   DATA[374,25] := 2.0;
   DATA[374,26] := 7.879262;
   DATA[374,27] := 144.7578;
   DATA[374,28] := 263.9067;
   DATA[374,29] := 12.03538;
   DATA[374,30] := 1.726096;
   DATA[374,31] := 1.271551;
   DATA[374,32] := 0.7345005;
   DATA[374,33] := 0.3086186;
   DATA[374,34] := 2.0;
   DATA[374,35] := 250.8972;
   DATA[374,36] := 1.617916;
   DATA[374,37] := 189.6789;
   DATA[374,38] := 0.000128152;
   DATA[374,39] := 1.0;
   DATA[375,0] := 2.625308;
   DATA[375,1] := 529.1664;
   DATA[375,2] := 2.0;
   DATA[375,3] := 2.0;
   DATA[375,4] := 262.0802;
   DATA[375,5] := 8.393553;
   DATA[375,6] := 328.0954;
   DATA[375,7] := 2.440265;
   DATA[375,8] := 2.0;
   DATA[375,9] := 2.0;
   DATA[375,10] := 2.0;
   DATA[375,11] := 19.73558;
   DATA[375,12] := 2.206322;
   DATA[375,13] := 971.9864;
   DATA[375,14] := 1.0;
   DATA[375,15] := 2.0;
   DATA[375,16] := 1.0;
   DATA[375,17] := 1.0;
   DATA[375,18] := 1.0;
   DATA[375,19] := 2.0;
   DATA[375,20] := 148.808;
   DATA[375,21] := 156.0369;
   DATA[375,22] := 1.719412;
   DATA[375,23] := 971.674;
   DATA[375,24] := 2.0;
   DATA[375,25] := 2.0;
   DATA[375,26] := 7.879262;
   DATA[375,27] := 144.7578;
   DATA[375,28] := 263.9067;
   DATA[375,29] := 12.03538;
   DATA[375,30] := 1.727634;
   DATA[375,31] := 1.287562;
   DATA[375,32] := 0.7345005;
   DATA[375,33] := 0.3086186;
   DATA[375,34] := 2.0;
   DATA[375,35] := 250.8972;
   DATA[375,36] := 1.617916;
   DATA[375,37] := 189.6789;
   DATA[375,38] := 0.000128152;
   DATA[375,39] := 1.0;
   DATA[376,0] := 2.619223;
   DATA[376,1] := 529.559;
   DATA[376,2] := 2.0;
   DATA[376,3] := 2.0;
   DATA[376,4] := 262.0802;
   DATA[376,5] := 8.393553;
   DATA[376,6] := 328.0954;
   DATA[376,7] := 2.440265;
   DATA[376,8] := 2.0;
   DATA[376,9] := 2.0;
   DATA[376,10] := 2.0;
   DATA[376,11] := 19.65875;
   DATA[376,12] := 2.206322;
   DATA[376,13] := 972.0665;
   DATA[376,14] := 1.0;
   DATA[376,15] := 2.0;
   DATA[376,16] := 1.0;
   DATA[376,17] := 1.0;
   DATA[376,18] := 1.0;
   DATA[376,19] := 2.0;
   DATA[376,20] := 148.808;
   DATA[376,21] := 156.0882;
   DATA[376,22] := 1.718002;
   DATA[376,23] := 971.3663;
   DATA[376,24] := 2.0;
   DATA[376,25] := 2.0;
   DATA[376,26] := 7.879262;
   DATA[376,27] := 144.7578;
   DATA[376,28] := 263.9067;
   DATA[376,29] := 12.03538;
   DATA[376,30] := 1.727634;
   DATA[376,31] := 1.301396;
   DATA[376,32] := 0.7353967;
   DATA[376,33] := 0.3086186;
   DATA[376,34] := 2.0;
   DATA[376,35] := 250.8972;
   DATA[376,36] := 1.617916;
   DATA[376,37] := 189.6629;
   DATA[376,38] := 0.000128152;
   DATA[376,39] := 1.0;
   DATA[377,0] := 2.612818;
   DATA[377,1] := 529.402;
   DATA[377,2] := 2.0;
   DATA[377,3] := 2.0;
   DATA[377,4] := 262.0802;
   DATA[377,5] := 8.393553;
   DATA[377,6] := 328.0954;
   DATA[377,7] := 2.440265;
   DATA[377,8] := 2.0;
   DATA[377,9] := 2.0;
   DATA[377,10] := 2.0;
   DATA[377,11] := 19.65875;
   DATA[377,12] := 2.208628;
   DATA[377,13] := 972.1466;
   DATA[377,14] := 1.0;
   DATA[377,15] := 2.0;
   DATA[377,16] := 1.0;
   DATA[377,17] := 1.0;
   DATA[377,18] := 1.0;
   DATA[377,19] := 2.0;
   DATA[377,20] := 148.808;
   DATA[377,21] := 156.1651;
   DATA[377,22] := 1.717874;
   DATA[377,23] := 971.251;
   DATA[377,24] := 2.0;
   DATA[377,25] := 2.0;
   DATA[377,26] := 7.879262;
   DATA[377,27] := 144.7578;
   DATA[377,28] := 263.9067;
   DATA[377,29] := 12.03538;
   DATA[377,30] := 1.727634;
   DATA[377,31] := 1.312028;
   DATA[377,32] := 0.7353967;
   DATA[377,33] := 0.3075297;
   DATA[377,34] := 2.0;
   DATA[377,35] := 250.8972;
   DATA[377,36] := 1.69801;
   DATA[377,37] := 189.5988;
   DATA[377,38] := 0.000128152;
   DATA[377,39] := 1.0;
   DATA[378,0] := 2.593601;
   DATA[378,1] := 529.7552;
   DATA[378,2] := 2.0;
   DATA[378,3] := 2.0;
   DATA[378,4] := 262.0802;
   DATA[378,5] := 8.393553;
   DATA[378,6] := 328.0954;
   DATA[378,7] := 2.440265;
   DATA[378,8] := 2.0;
   DATA[378,9] := 2.0;
   DATA[378,10] := 2.0;
   DATA[378,11] := 19.65875;
   DATA[378,12] := 2.209013;
   DATA[378,13] := 972.467;
   DATA[378,14] := 1.0;
   DATA[378,15] := 2.0;
   DATA[378,16] := 1.0;
   DATA[378,17] := 1.0;
   DATA[378,18] := 1.0;
   DATA[378,19] := 2.0;
   DATA[378,20] := 148.808;
   DATA[378,21] := 156.1651;
   DATA[378,22] := 1.716592;
   DATA[378,23] := 971.1741;
   DATA[378,24] := 2.0;
   DATA[378,25] := 2.0;
   DATA[378,26] := 7.879262;
   DATA[378,27] := 144.7578;
   DATA[378,28] := 263.9067;
   DATA[378,29] := 12.03538;
   DATA[378,30] := 1.727634;
   DATA[378,31] := 1.312284;
   DATA[378,32] := 0.7353967;
   DATA[378,33] := 0.306761;
   DATA[378,34] := 2.0;
   DATA[378,35] := 250.8972;
   DATA[378,36] := 1.69801;
   DATA[378,37] := 189.4386;
   DATA[378,38] := 0.000128152;
   DATA[378,39] := 1.0;
   DATA[379,0] := 2.578868;
   DATA[379,1] := 529.9907;
   DATA[379,2] := 2.0;
   DATA[379,3] := 2.0;
   DATA[379,4] := 262.0802;
   DATA[379,5] := 8.393553;
   DATA[379,6] := 328.0954;
   DATA[379,7] := 2.440265;
   DATA[379,8] := 2.0;
   DATA[379,9] := 2.0;
   DATA[379,10] := 2.0;
   DATA[379,11] := 19.72598;
   DATA[379,12] := 2.209269;
   DATA[379,13] := 972.467;
   DATA[379,14] := 1.0;
   DATA[379,15] := 2.0;
   DATA[379,16] := 1.0;
   DATA[379,17] := 1.0;
   DATA[379,18] := 1.0;
   DATA[379,19] := 2.0;
   DATA[379,20] := 148.808;
   DATA[379,21] := 156.1651;
   DATA[379,22] := 1.715439;
   DATA[379,23] := 971.4817;
   DATA[379,24] := 2.0;
   DATA[379,25] := 2.0;
   DATA[379,26] := 7.879262;
   DATA[379,27] := 144.7578;
   DATA[379,28] := 263.7465;
   DATA[379,29] := 12.03538;
   DATA[379,30] := 1.726737;
   DATA[379,31] := 1.296016;
   DATA[379,32] := 0.7353967;
   DATA[379,33] := 0.3086186;
   DATA[379,34] := 2.0;
   DATA[379,35] := 250.8972;
   DATA[379,36] := 1.69801;
   DATA[379,37] := 189.4386;
   DATA[379,38] := 0.000128152;
   DATA[379,39] := 1.0;
   DATA[380,0] := 2.561253;
   DATA[380,1] := 530.4225;
   DATA[380,2] := 2.0;
   DATA[380,3] := 2.0;
   DATA[380,4] := 262.0802;
   DATA[380,5] := 8.393553;
   DATA[380,6] := 328.0954;
   DATA[380,7] := 2.440265;
   DATA[380,8] := 2.0;
   DATA[380,9] := 2.0;
   DATA[380,10] := 2.0;
   DATA[380,11] := 19.72598;
   DATA[380,12] := 2.211959;
   DATA[380,13] := 972.7474;
   DATA[380,14] := 1.0;
   DATA[380,15] := 2.0;
   DATA[380,16] := 1.0;
   DATA[380,17] := 1.0;
   DATA[380,18] := 1.0;
   DATA[380,19] := 2.0;
   DATA[380,20] := 148.808;
   DATA[380,21] := 156.1651;
   DATA[380,22] := 1.71467;
   DATA[380,23] := 971.674;
   DATA[380,24] := 2.0;
   DATA[380,25] := 2.0;
   DATA[380,26] := 7.879262;
   DATA[380,27] := 144.7578;
   DATA[380,28] := 263.7465;
   DATA[380,29] := 12.03538;
   DATA[380,30] := 1.726737;
   DATA[380,31] := 1.284745;
   DATA[380,32] := 0.7353967;
   DATA[380,33] := 0.3086186;
   DATA[380,34] := 2.0;
   DATA[380,35] := 250.737;
   DATA[380,36] := 1.69801;
   DATA[380,37] := 189.4386;
   DATA[380,38] := 0.000128152;
   DATA[380,39] := 1.0;
   DATA[381,0] := 2.541716;
   DATA[381,1] := 530.187;
   DATA[381,2] := 2.0;
   DATA[381,3] := 2.0;
   DATA[381,4] := 262.0802;
   DATA[381,5] := 8.393553;
   DATA[381,6] := 328.0954;
   DATA[381,7] := 2.440265;
   DATA[381,8] := 2.0;
   DATA[381,9] := 2.0;
   DATA[381,10] := 2.0;
   DATA[381,11] := 19.72598;
   DATA[381,12] := 2.211959;
   DATA[381,13] := 972.6273;
   DATA[381,14] := 1.0;
   DATA[381,15] := 2.0;
   DATA[381,16] := 1.0;
   DATA[381,17] := 1.0;
   DATA[381,18] := 1.0;
   DATA[381,19] := 2.0;
   DATA[381,20] := 148.808;
   DATA[381,21] := 156.1651;
   DATA[381,22] := 1.714286;
   DATA[381,23] := 971.674;
   DATA[381,24] := 2.0;
   DATA[381,25] := 2.0;
   DATA[381,26] := 7.879262;
   DATA[381,27] := 144.7578;
   DATA[381,28] := 263.7465;
   DATA[381,29] := 12.03538;
   DATA[381,30] := 1.726737;
   DATA[381,31] := 1.282567;
   DATA[381,32] := 0.7353967;
   DATA[381,33] := 0.3075937;
   DATA[381,34] := 2.0;
   DATA[381,35] := 250.737;
   DATA[381,36] := 1.69801;
   DATA[381,37] := 189.4386;
   DATA[381,38] := 0.000128152;
   DATA[381,39] := 1.0;
   DATA[382,0] := 2.527303;
   DATA[382,1] := 530.501;
   DATA[382,2] := 2.0;
   DATA[382,3] := 2.0;
   DATA[382,4] := 262.0802;
   DATA[382,5] := 8.393553;
   DATA[382,6] := 328.2235;
   DATA[382,7] := 2.440265;
   DATA[382,8] := 2.0;
   DATA[382,9] := 2.0;
   DATA[382,10] := 2.0;
   DATA[382,11] := 19.72598;
   DATA[382,12] := 2.211959;
   DATA[382,13] := 972.5872;
   DATA[382,14] := 1.0;
   DATA[382,15] := 2.0;
   DATA[382,16] := 1.0;
   DATA[382,17] := 1.0;
   DATA[382,18] := 1.0;
   DATA[382,19] := 2.0;
   DATA[382,20] := 148.808;
   DATA[382,21] := 155.9856;
   DATA[382,22] := 1.713517;
   DATA[382,23] := 971.674;
   DATA[382,24] := 2.0;
   DATA[382,25] := 2.0;
   DATA[382,26] := 7.879262;
   DATA[382,27] := 144.7578;
   DATA[382,28] := 263.7465;
   DATA[382,29] := 12.03538;
   DATA[382,30] := 1.726737;
   DATA[382,31] := 1.296273;
   DATA[382,32] := 0.7353967;
   DATA[382,33] := 0.3068251;
   DATA[382,34] := 2.0;
   DATA[382,35] := 250.737;
   DATA[382,36] := 1.681991;
   DATA[382,37] := 189.4386;
   DATA[382,38] := 0.000128152;
   DATA[382,39] := 1.0;
   DATA[383,0] := 2.506485;
   DATA[383,1] := 530.3832;
   DATA[383,2] := 2.0;
   DATA[383,3] := 2.0;
   DATA[383,4] := 262.0802;
   DATA[383,5] := 8.393553;
   DATA[383,6] := 328.2235;
   DATA[383,7] := 2.440265;
   DATA[383,8] := 2.0;
   DATA[383,9] := 2.0;
   DATA[383,10] := 2.0;
   DATA[383,11] := 19.69396;
   DATA[383,12] := 2.211959;
   DATA[383,13] := 972.8676;
   DATA[383,14] := 1.0;
   DATA[383,15] := 2.0;
   DATA[383,16] := 1.0;
   DATA[383,17] := 1.0;
   DATA[383,18] := 1.0;
   DATA[383,19] := 2.0;
   DATA[383,20] := 148.808;
   DATA[383,21] := 155.9856;
   DATA[383,22] := 1.715824;
   DATA[383,23] := 971.8662;
   DATA[383,24] := 2.0;
   DATA[383,25] := 2.0;
   DATA[383,26] := 7.879262;
   DATA[383,27] := 144.7578;
   DATA[383,28] := 263.7465;
   DATA[383,29] := 12.03538;
   DATA[383,30] := 1.726737;
   DATA[383,31] := 1.30114;
   DATA[383,32] := 0.7353967;
   DATA[383,33] := 0.3068251;
   DATA[383,34] := 2.0;
   DATA[383,35] := 250.737;
   DATA[383,36] := 1.681991;
   DATA[383,37] := 189.5027;
   DATA[383,38] := 0.000128152;
   DATA[383,39] := 1.0;
   DATA[384,0] := 2.493995;
   DATA[384,1] := 530.4225;
   DATA[384,2] := 2.0;
   DATA[384,3] := 2.0;
   DATA[384,4] := 262.0802;
   DATA[384,5] := 8.393553;
   DATA[384,6] := 328.2235;
   DATA[384,7] := 2.440265;
   DATA[384,8] := 2.0;
   DATA[384,9] := 2.0;
   DATA[384,10] := 2.0;
   DATA[384,11] := 19.69396;
   DATA[384,12] := 2.211959;
   DATA[384,13] := 972.8275;
   DATA[384,14] := 1.0;
   DATA[384,15] := 2.0;
   DATA[384,16] := 1.0;
   DATA[384,17] := 1.0;
   DATA[384,18] := 1.0;
   DATA[384,19] := 2.0;
   DATA[384,20] := 148.808;
   DATA[384,21] := 155.9856;
   DATA[384,22] := 1.71813;
   DATA[384,23] := 971.674;
   DATA[384,24] := 2.0;
   DATA[384,25] := 2.0;
   DATA[384,26] := 7.879262;
   DATA[384,27] := 144.7578;
   DATA[384,28] := 263.7465;
   DATA[384,29] := 12.03538;
   DATA[384,30] := 1.726737;
   DATA[384,31] := 1.292174;
   DATA[384,32] := 0.7353967;
   DATA[384,33] := 0.3063127;
   DATA[384,34] := 2.0;
   DATA[384,35] := 250.8972;
   DATA[384,36] := 1.681991;
   DATA[384,37] := 189.5668;
   DATA[384,38] := 0.000128152;
   DATA[384,39] := 1.0;
   DATA[385,0] := 2.477981;
   DATA[385,1] := 529.9122;
   DATA[385,2] := 2.0;
   DATA[385,3] := 2.0;
   DATA[385,4] := 262.0802;
   DATA[385,5] := 8.390669;
   DATA[385,6] := 328.2235;
   DATA[385,7] := 2.440265;
   DATA[385,8] := 2.0;
   DATA[385,9] := 2.0;
   DATA[385,10] := 2.0;
   DATA[385,11] := 19.65555;
   DATA[385,12] := 2.212343;
   DATA[385,13] := 973.188;
   DATA[385,14] := 1.0;
   DATA[385,15] := 2.0;
   DATA[385,16] := 1.0;
   DATA[385,17] := 1.0;
   DATA[385,18] := 1.0;
   DATA[385,19] := 2.0;
   DATA[385,20] := 148.808;
   DATA[385,21] := 155.9856;
   DATA[385,22] := 1.71813;
   DATA[385,23] := 971.7509;
   DATA[385,24] := 2.0;
   DATA[385,25] := 2.0;
   DATA[385,26] := 7.879262;
   DATA[385,27] := 144.7578;
   DATA[385,28] := 263.7465;
   DATA[385,29] := 12.30454;
   DATA[385,30] := 1.726737;
   DATA[385,31] := 1.285001;
   DATA[385,32] := 0.7353967;
   DATA[385,33] := 0.3063127;
   DATA[385,34] := 2.0;
   DATA[385,35] := 250.9453;
   DATA[385,36] := 1.681991;
   DATA[385,37] := 189.5668;
   DATA[385,38] := 0.000128152;
   DATA[385,39] := 1.0;
   DATA[386,0] := 2.46549;
   DATA[386,1] := 529.7159;
   DATA[386,2] := 2.0;
   DATA[386,3] := 2.0;
   DATA[386,4] := 262.0802;
   DATA[386,5] := 8.390669;
   DATA[386,6] := 328.2235;
   DATA[386,7] := 2.440265;
   DATA[386,8] := 2.0;
   DATA[386,9] := 2.0;
   DATA[386,10] := 2.0;
   DATA[386,11] := 19.65555;
   DATA[386,12] := 2.212343;
   DATA[386,13] := 973.2681;
   DATA[386,14] := 1.0;
   DATA[386,15] := 2.0;
   DATA[386,16] := 1.0;
   DATA[386,17] := 1.0;
   DATA[386,18] := 1.0;
   DATA[386,19] := 2.0;
   DATA[386,20] := 148.808;
   DATA[386,21] := 155.9856;
   DATA[386,22] := 1.71813;
   DATA[386,23] := 971.9431;
   DATA[386,24] := 2.0;
   DATA[386,25] := 2.0;
   DATA[386,26] := 7.879262;
   DATA[386,27] := 144.7578;
   DATA[386,28] := 263.7465;
   DATA[386,29] := 12.30454;
   DATA[386,30] := 1.726737;
   DATA[386,31] := 1.27232;
   DATA[386,32] := 0.7353967;
   DATA[386,33] := 0.3068891;
   DATA[386,34] := 2.0;
   DATA[386,35] := 250.9453;
   DATA[386,36] := 1.681991;
   DATA[386,37] := 189.6949;
   DATA[386,38] := 0.000128152;
   DATA[386,39] := 1.0;
   DATA[387,0] := 2.449156;
   DATA[387,1] := 529.3234;
   DATA[387,2] := 2.0;
   DATA[387,3] := 2.0;
   DATA[387,4] := 262.0802;
   DATA[387,5] := 8.390669;
   DATA[387,6] := 328.2235;
   DATA[387,7] := 2.440265;
   DATA[387,8] := 2.0;
   DATA[387,9] := 2.0;
   DATA[387,10] := 2.0;
   DATA[387,11] := 19.65555;
   DATA[387,12] := 2.212343;
   DATA[387,13] := 973.4283;
   DATA[387,14] := 1.0;
   DATA[387,15] := 2.0;
   DATA[387,16] := 1.0;
   DATA[387,17] := 1.0;
   DATA[387,18] := 1.0;
   DATA[387,19] := 2.0;
   DATA[387,20] := 148.808;
   DATA[387,21] := 155.9856;
   DATA[387,22] := 1.71813;
   DATA[387,23] := 971.8662;
   DATA[387,24] := 2.0;
   DATA[387,25] := 2.0;
   DATA[387,26] := 7.87766;
   DATA[387,27] := 144.7578;
   DATA[387,28] := 263.7465;
   DATA[387,29] := 12.15073;
   DATA[387,30] := 1.726737;
   DATA[387,31] := 1.271551;
   DATA[387,32] := 0.7353967;
   DATA[387,33] := 0.3068891;
   DATA[387,34] := 2.0;
   DATA[387,35] := 251.0414;
   DATA[387,36] := 1.681991;
   DATA[387,37] := 189.6949;
   DATA[387,38] := 0.000128152;
   DATA[387,39] := 1.0;
   DATA[388,0] := 2.436345;
   DATA[388,1] := 528.9309;
   DATA[388,2] := 2.0;
   DATA[388,3] := 2.0;
   DATA[388,4] := 262.0802;
   DATA[388,5] := 8.390669;
   DATA[388,6] := 328.2235;
   DATA[388,7] := 2.440265;
   DATA[388,8] := 2.0;
   DATA[388,9] := 2.0;
   DATA[388,10] := 2.0;
   DATA[388,11] := 19.58832;
   DATA[388,12] := 2.212984;
   DATA[388,13] := 973.6686;
   DATA[388,14] := 1.0;
   DATA[388,15] := 2.0;
   DATA[388,16] := 1.0;
   DATA[388,17] := 1.0;
   DATA[388,18] := 1.0;
   DATA[388,19] := 2.0;
   DATA[388,20] := 148.808;
   DATA[388,21] := 155.9856;
   DATA[388,22] := 1.71813;
   DATA[388,23] := 971.9047;
   DATA[388,24] := 2.0;
   DATA[388,25] := 2.0;
   DATA[388,26] := 7.87766;
   DATA[388,27] := 144.7578;
   DATA[388,28] := 263.7465;
   DATA[388,29] := 12.15073;
   DATA[388,30] := 1.726737;
   DATA[388,31] := 1.271551;
   DATA[388,32] := 0.7353967;
   DATA[388,33] := 0.3068891;
   DATA[388,34] := 2.0;
   DATA[388,35] := 251.1055;
   DATA[388,36] := 1.681991;
   DATA[388,37] := 189.6949;
   DATA[388,38] := 0.000128152;
   DATA[388,39] := 1.0;
   DATA[389,0] := 2.425456;
   DATA[389,1] := 528.7347;
   DATA[389,2] := 2.0;
   DATA[389,3] := 2.0;
   DATA[389,4] := 262.0802;
   DATA[389,5] := 8.390669;
   DATA[389,6] := 328.2235;
   DATA[389,7] := 2.440265;
   DATA[389,8] := 2.0;
   DATA[389,9] := 2.0;
   DATA[389,10] := 2.0;
   DATA[389,11] := 19.57872;
   DATA[389,12] := 2.212984;
   DATA[389,13] := 974.1893;
   DATA[389,14] := 1.0;
   DATA[389,15] := 2.0;
   DATA[389,16] := 1.0;
   DATA[389,17] := 1.0;
   DATA[389,18] := 1.0;
   DATA[389,19] := 2.0;
   DATA[389,20] := 148.808;
   DATA[389,21] := 155.9856;
   DATA[389,22] := 1.719924;
   DATA[389,23] := 972.2892;
   DATA[389,24] := 2.0;
   DATA[389,25] := 2.0;
   DATA[389,26] := 7.87766;
   DATA[389,27] := 144.7578;
   DATA[389,28] := 263.7465;
   DATA[389,29] := 12.07383;
   DATA[389,30] := 1.726737;
   DATA[389,31] := 1.285513;
   DATA[389,32] := 0.7353967;
   DATA[389,33] := 0.3068891;
   DATA[389,34] := 2.0;
   DATA[389,35] := 251.1055;
   DATA[389,36] := 1.681991;
   DATA[389,37] := 189.8391;
   DATA[389,38] := 0.000128152;
   DATA[389,39] := 1.0;
   DATA[390,0] := 2.420651;
   DATA[390,1] := 528.6561;
   DATA[390,2] := 2.0;
   DATA[390,3] := 2.0;
   DATA[390,4] := 262.0802;
   DATA[390,5] := 8.390669;
   DATA[390,6] := 328.0441;
   DATA[390,7] := 2.440265;
   DATA[390,8] := 2.0;
   DATA[390,9] := 2.0;
   DATA[390,10] := 2.0;
   DATA[390,11] := 19.57872;
   DATA[390,12] := 2.212984;
   DATA[390,13] := 974.2695;
   DATA[390,14] := 1.0;
   DATA[390,15] := 2.0;
   DATA[390,16] := 1.0;
   DATA[390,17] := 1.0;
   DATA[390,18] := 1.0;
   DATA[390,19] := 2.0;
   DATA[390,20] := 148.808;
   DATA[390,21] := 155.9856;
   DATA[390,22] := 1.719924;
   DATA[390,23] := 972.5967;
   DATA[390,24] := 2.0;
   DATA[390,25] := 2.0;
   DATA[390,26] := 7.87766;
   DATA[390,27] := 144.7578;
   DATA[390,28] := 263.7465;
   DATA[390,29] := 12.03538;
   DATA[390,30] := 1.726737;
   DATA[390,31] := 1.302165;
   DATA[390,32] := 0.7353967;
   DATA[390,33] := 0.3068891;
   DATA[390,34] := 2.0;
   DATA[390,35] := 251.1055;
   DATA[390,36] := 1.681991;
   DATA[390,37] := 189.8391;
   DATA[390,38] := 0.000128152;
   DATA[390,39] := 1.0;
   DATA[391,0] := 2.428338;
   DATA[391,1] := 528.3421;
   DATA[391,2] := 2.0;
   DATA[391,3] := 2.0;
   DATA[391,4] := 262.0802;
   DATA[391,5] := 8.390669;
   DATA[391,6] := 328.0441;
   DATA[391,7] := 2.440265;
   DATA[391,8] := 2.0;
   DATA[391,9] := 2.0;
   DATA[391,10] := 2.0;
   DATA[391,11] := 19.57872;
   DATA[391,12] := 2.212984;
   DATA[391,13] := 973.7487;
   DATA[391,14] := 1.0;
   DATA[391,15] := 2.0;
   DATA[391,16] := 1.0;
   DATA[391,17] := 1.0;
   DATA[391,18] := 1.0;
   DATA[391,19] := 2.0;
   DATA[391,20] := 148.808;
   DATA[391,21] := 155.9856;
   DATA[391,22] := 1.719027;
   DATA[391,23] := 972.2892;
   DATA[391,24] := 2.0;
   DATA[391,25] := 2.0;
   DATA[391,26] := 7.87766;
   DATA[391,27] := 144.7578;
   DATA[391,28] := 263.7465;
   DATA[391,29] := 12.03538;
   DATA[391,30] := 1.726737;
   DATA[391,31] := 1.32932;
   DATA[391,32] := 0.7353967;
   DATA[391,33] := 0.3061845;
   DATA[391,34] := 2.0;
   DATA[391,35] := 251.1055;
   DATA[391,36] := 1.681991;
   DATA[391,37] := 189.8391;
   DATA[391,38] := 0.000128152;
   DATA[391,39] := 1.0;
   DATA[392,0] := 2.474778;
   DATA[392,1] := 528.0674;
   DATA[392,2] := 2.0;
   DATA[392,3] := 2.0;
   DATA[392,4] := 262.0802;
   DATA[392,5] := 8.39163;
   DATA[392,6] := 328.0441;
   DATA[392,7] := 2.440265;
   DATA[392,8] := 2.0;
   DATA[392,9] := 2.0;
   DATA[392,10] := 2.0;
   DATA[392,11] := 19.57872;
   DATA[392,12] := 2.212984;
   DATA[392,13] := 973.4684;
   DATA[392,14] := 1.0;
   DATA[392,15] := 2.0;
   DATA[392,16] := 1.0;
   DATA[392,17] := 1.0;
   DATA[392,18] := 1.0;
   DATA[392,19] := 2.0;
   DATA[392,20] := 148.808;
   DATA[392,21] := 155.9856;
   DATA[392,22] := 1.71813;
   DATA[392,23] := 972.2507;
   DATA[392,24] := 2.0;
   DATA[392,25] := 2.0;
   DATA[392,26] := 7.87766;
   DATA[392,27] := 144.8347;
   DATA[392,28] := 263.7465;
   DATA[392,29] := 12.03538;
   DATA[392,30] := 1.726737;
   DATA[392,31] := 1.332266;
   DATA[392,32] := 0.7353967;
   DATA[392,33] := 0.3070813;
   DATA[392,34] := 2.0;
   DATA[392,35] := 251.1055;
   DATA[392,36] := 1.681991;
   DATA[392,37] := 189.8391;
   DATA[392,38] := 0.000128152;
   DATA[392,39] := 1.0;
   DATA[393,0] := 2.524101;
   DATA[393,1] := 528.1459;
   DATA[393,2] := 2.0;
   DATA[393,3] := 2.0;
   DATA[393,4] := 262.0802;
   DATA[393,5] := 8.39163;
   DATA[393,6] := 328.0441;
   DATA[393,7] := 2.440265;
   DATA[393,8] := 2.0;
   DATA[393,9] := 2.0;
   DATA[393,10] := 2.0;
   DATA[393,11] := 19.66195;
   DATA[393,12] := 2.212984;
   DATA[393,13] := 973.7487;
   DATA[393,14] := 1.0;
   DATA[393,15] := 2.0;
   DATA[393,16] := 1.0;
   DATA[393,17] := 1.0;
   DATA[393,18] := 1.0;
   DATA[393,19] := 2.0;
   DATA[393,20] := 148.808;
   DATA[393,21] := 155.9856;
   DATA[393,22] := 1.71813;
   DATA[393,23] := 972.3276;
   DATA[393,24] := 2.0;
   DATA[393,25] := 2.0;
   DATA[393,26] := 7.87766;
   DATA[393,27] := 144.8603;
   DATA[393,28] := 263.7465;
   DATA[393,29] := 12.03538;
   DATA[393,30] := 1.728147;
   DATA[393,31] := 1.325221;
   DATA[393,32] := 0.7353967;
   DATA[393,33] := 0.3070813;
   DATA[393,34] := 2.0;
   DATA[393,35] := 251.1055;
   DATA[393,36] := 1.681991;
   DATA[393,37] := 189.6469;
   DATA[393,38] := 0.000128152;
   DATA[393,39] := 1.0;
   DATA[394,0] := 2.552285;
   DATA[394,1] := 527.7926;
   DATA[394,2] := 2.0;
   DATA[394,3] := 2.0;
   DATA[394,4] := 262.0802;
   DATA[394,5] := 8.39163;
   DATA[394,6] := 328.0441;
   DATA[394,7] := 2.440265;
   DATA[394,8] := 2.0;
   DATA[394,9] := 2.0;
   DATA[394,10] := 2.0;
   DATA[394,11] := 19.66195;
   DATA[394,12] := 2.212343;
   DATA[394,13] := 973.3882;
   DATA[394,14] := 1.0;
   DATA[394,15] := 2.0;
   DATA[394,16] := 1.0;
   DATA[394,17] := 1.0;
   DATA[394,18] := 1.0;
   DATA[394,19] := 2.0;
   DATA[394,20] := 148.808;
   DATA[394,21] := 155.7293;
   DATA[394,22] := 1.71813;
   DATA[394,23] := 972.0585;
   DATA[394,24] := 2.0;
   DATA[394,25] := 2.0;
   DATA[394,26] := 7.87766;
   DATA[394,27] := 144.8603;
   DATA[394,28] := 263.7465;
   DATA[394,29] := 12.03538;
   DATA[394,30] := 1.728147;
   DATA[394,31] := 1.315614;
   DATA[394,32] := 0.7353967;
   DATA[394,33] := 0.3070813;
   DATA[394,34] := 2.0;
   DATA[394,35] := 251.1055;
   DATA[394,36] := 1.681991;
   DATA[394,37] := 189.6469;
   DATA[394,38] := 0.000128152;
   DATA[394,39] := 1.0;
   DATA[395,0] := 2.593921;
   DATA[395,1] := 527.9496;
   DATA[395,2] := 2.0;
   DATA[395,3] := 2.0;
   DATA[395,4] := 262.0802;
   DATA[395,5] := 8.393873;
   DATA[395,6] := 328.0441;
   DATA[395,7] := 2.436933;
   DATA[395,8] := 2.0;
   DATA[395,9] := 2.0;
   DATA[395,10] := 2.0;
   DATA[395,11] := 19.66195;
   DATA[395,12] := 2.210678;
   DATA[395,13] := 973.949;
   DATA[395,14] := 1.0;
   DATA[395,15] := 2.0;
   DATA[395,16] := 1.0;
   DATA[395,17] := 1.0;
   DATA[395,18] := 1.0;
   DATA[395,19] := 2.0;
   DATA[395,20] := 148.808;
   DATA[395,21] := 155.7293;
   DATA[395,22] := 1.71813;
   DATA[395,23] := 972.0969;
   DATA[395,24] := 2.0;
   DATA[395,25] := 2.0;
   DATA[395,26] := 7.87798;
   DATA[395,27] := 144.8603;
   DATA[395,28] := 263.7465;
   DATA[395,29] := 12.15073;
   DATA[395,30] := 1.728531;
   DATA[395,31] := 1.285769;
   DATA[395,32] := 0.7353967;
   DATA[395,33] := 0.3084905;
   DATA[395,34] := 2.0;
   DATA[395,35] := 251.1055;
   DATA[395,36] := 1.681991;
   DATA[395,37] := 189.6469;
   DATA[395,38] := 0.000128152;
   DATA[395,39] := 1.0;
   DATA[396,0] := 2.621785;
   DATA[396,1] := 527.7534;
   DATA[396,2] := 2.0;
   DATA[396,3] := 2.0;
   DATA[396,4] := 262.0802;
   DATA[396,5] := 8.393873;
   DATA[396,6] := 328.0441;
   DATA[396,7] := 2.436933;
   DATA[396,8] := 2.0;
   DATA[396,9] := 2.0;
   DATA[396,10] := 2.0;
   DATA[396,11] := 19.71637;
   DATA[396,12] := 2.210037;
   DATA[396,13] := 974.0692;
   DATA[396,14] := 1.0;
   DATA[396,15] := 2.0;
   DATA[396,16] := 1.0;
   DATA[396,17] := 1.0;
   DATA[396,18] := 1.0;
   DATA[396,19] := 2.0;
   DATA[396,20] := 148.808;
   DATA[396,21] := 155.7293;
   DATA[396,22] := 1.71813;
   DATA[396,23] := 972.4045;
   DATA[396,24] := 2.0;
   DATA[396,25] := 2.0;
   DATA[396,26] := 7.879582;
   DATA[396,27] := 144.8603;
   DATA[396,28] := 263.7465;
   DATA[396,29] := 12.15073;
   DATA[396,30] := 1.728788;
   DATA[396,31] := 1.26758;
   DATA[396,32] := 0.7353967;
   DATA[396,33] := 0.3075297;
   DATA[396,34] := 2.0;
   DATA[396,35] := 250.9933;
   DATA[396,36] := 1.681991;
   DATA[396,37] := 189.6469;
   DATA[396,38] := 0.000128152;
   DATA[396,39] := 1.0;
   DATA[397,0] := 2.654774;
   DATA[397,1] := 527.6356;
   DATA[397,2] := 2.0;
   DATA[397,3] := 2.0;
   DATA[397,4] := 262.0802;
   DATA[397,5] := 8.393873;
   DATA[397,6] := 328.0441;
   DATA[397,7] := 2.440265;
   DATA[397,8] := 2.0;
   DATA[397,9] := 2.0;
   DATA[397,10] := 2.0;
   DATA[397,11] := 19.71637;
   DATA[397,12] := 2.210037;
   DATA[397,13] := 974.2695;
   DATA[397,14] := 1.0;
   DATA[397,15] := 2.0;
   DATA[397,16] := 1.0;
   DATA[397,17] := 1.0;
   DATA[397,18] := 1.0;
   DATA[397,19] := 2.0;
   DATA[397,20] := 148.808;
   DATA[397,21] := 155.7293;
   DATA[397,22] := 1.71813;
   DATA[397,23] := 972.443;
   DATA[397,24] := 2.0;
   DATA[397,25] := 2.0;
   DATA[397,26] := 7.879582;
   DATA[397,27] := 144.8603;
   DATA[397,28] := 263.7465;
   DATA[397,29] := 12.15073;
   DATA[397,30] := 1.729172;
   DATA[397,31] := 1.265147;
   DATA[397,32] := 0.7353967;
   DATA[397,33] := 0.3081703;
   DATA[397,34] := 2.0;
   DATA[397,35] := 250.8972;
   DATA[397,36] := 1.681991;
   DATA[397,37] := 189.6469;
   DATA[397,38] := 0.000128152;
   DATA[397,39] := 1.0;
   DATA[398,0] := 2.666944;
   DATA[398,1] := 527.8711;
   DATA[398,2] := 2.0;
   DATA[398,3] := 2.0;
   DATA[398,4] := 262.0802;
   DATA[398,5] := 8.393873;
   DATA[398,6] := 328.0441;
   DATA[398,7] := 2.440265;
   DATA[398,8] := 2.0;
   DATA[398,9] := 2.0;
   DATA[398,10] := 2.0;
   DATA[398,11] := 19.71637;
   DATA[398,12] := 2.210037;
   DATA[398,13] := 974.8702;
   DATA[398,14] := 1.0;
   DATA[398,15] := 2.0;
   DATA[398,16] := 1.0;
   DATA[398,17] := 1.0;
   DATA[398,18] := 1.0;
   DATA[398,19] := 2.0;
   DATA[398,20] := 148.808;
   DATA[398,21] := 155.7293;
   DATA[398,22] := 1.71813;
   DATA[398,23] := 972.6736;
   DATA[398,24] := 2.0;
   DATA[398,25] := 2.0;
   DATA[398,26] := 7.879582;
   DATA[398,27] := 144.8603;
   DATA[398,28] := 263.7465;
   DATA[398,29] := 12.15073;
   DATA[398,30] := 1.729172;
   DATA[398,31] := 1.280902;
   DATA[398,32] := 0.7353967;
   DATA[398,33] := 0.3087468;
   DATA[398,34] := 2.0;
   DATA[398,35] := 250.8972;
   DATA[398,36] := 1.681991;
   DATA[398,37] := 189.6469;
   DATA[398,38] := 0.000128152;
   DATA[398,39] := 1.0;
   DATA[399,0] := 2.659258;
   DATA[399,1] := 528.1459;
   DATA[399,2] := 2.0;
   DATA[399,3] := 2.0;
   DATA[399,4] := 262.0802;
   DATA[399,5] := 8.393873;
   DATA[399,6] := 328.0441;
   DATA[399,7] := 2.440265;
   DATA[399,8] := 2.0;
   DATA[399,9] := 2.0;
   DATA[399,10] := 2.0;
   DATA[399,11] := 19.68756;
   DATA[399,12] := 2.210037;
   DATA[399,13] := 974.8302;
   DATA[399,14] := 1.0;
   DATA[399,15] := 2.0;
   DATA[399,16] := 1.0;
   DATA[399,17] := 1.0;
   DATA[399,18] := 1.0;
   DATA[399,19] := 2.0;
   DATA[399,20] := 148.808;
   DATA[399,21] := 155.7293;
   DATA[399,22] := 1.716849;
   DATA[399,23] := 972.9813;
   DATA[399,24] := 2.0;
   DATA[399,25] := 2.0;
   DATA[399,26] := 7.879582;
   DATA[399,27] := 144.8603;
   DATA[399,28] := 263.7465;
   DATA[399,29] := 12.15073;
   DATA[399,30] := 1.729172;
   DATA[399,31] := 1.291149;
   DATA[399,32] := 0.7353967;
   DATA[399,33] := 0.3077219;
   DATA[399,34] := 2.0;
   DATA[399,35] := 251.0254;
   DATA[399,36] := 1.681991;
   DATA[399,37] := 189.6469;
   DATA[399,38] := 0.000128152;
   DATA[399,39] := 1.0;
   DATA[400,0] := 2.637158;
   DATA[400,1] := 527.9496;
   DATA[400,2] := 2.0;
   DATA[400,3] := 2.0;
   DATA[400,4] := 262.0802;
   DATA[400,5] := 8.393873;
   DATA[400,6] := 328.0441;
   DATA[400,7] := 2.440265;
   DATA[400,8] := 2.0;
   DATA[400,9] := 2.0;
   DATA[400,10] := 2.0;
   DATA[400,11] := 19.61393;
   DATA[400,12] := 2.209269;
   DATA[400,13] := 975.1506;
   DATA[400,14] := 1.0;
   DATA[400,15] := 2.0;
   DATA[400,16] := 1.0;
   DATA[400,17] := 1.0;
   DATA[400,18] := 1.0;
   DATA[400,19] := 2.0;
   DATA[400,20] := 148.808;
   DATA[400,21] := 155.7293;
   DATA[400,22] := 1.716849;
   DATA[400,23] := 973.2889;
   DATA[400,24] := 2.0;
   DATA[400,25] := 2.0;
   DATA[400,26] := 7.879582;
   DATA[400,27] := 144.8603;
   DATA[400,28] := 263.7465;
   DATA[400,29] := 12.15073;
   DATA[400,30] := 1.729172;
   DATA[400,31] := 1.306648;
   DATA[400,32] := 0.736421;
   DATA[400,33] := 0.3068891;
   DATA[400,34] := 2.0;
   DATA[400,35] := 251.0254;
   DATA[400,36] := 1.681991;
   DATA[400,37] := 189.727;
   DATA[400,38] := 0.000128152;
   DATA[400,39] := 1.0;
   DATA[401,0] := 2.622426;
   DATA[401,1] := 527.6748;
   DATA[401,2] := 2.0;
   DATA[401,3] := 2.0;
   DATA[401,4] := 262.0802;
   DATA[401,5] := 8.393873;
   DATA[401,6] := 328.0441;
   DATA[401,7] := 2.441803;
   DATA[401,8] := 2.0;
   DATA[401,9] := 2.0;
   DATA[401,10] := 2.0;
   DATA[401,11] := 19.55311;
   DATA[401,12] := 2.209269;
   DATA[401,13] := 975.431;
   DATA[401,14] := 1.0;
   DATA[401,15] := 2.0;
   DATA[401,16] := 1.0;
   DATA[401,17] := 1.0;
   DATA[401,18] := 1.0;
   DATA[401,19] := 2.0;
   DATA[401,20] := 148.808;
   DATA[401,21] := 155.7293;
   DATA[401,22] := 1.716849;
   DATA[401,23] := 973.2889;
   DATA[401,24] := 2.0;
   DATA[401,25] := 2.0;
   DATA[401,26] := 7.879582;
   DATA[401,27] := 144.8603;
   DATA[401,28] := 263.7465;
   DATA[401,29] := 12.15073;
   DATA[401,30] := 1.729172;
   DATA[401,31] := 1.305495;
   DATA[401,32] := 0.736421;
   DATA[401,33] := 0.3066329;
   DATA[401,34] := 2.0;
   DATA[401,35] := 251.1055;
   DATA[401,36] := 1.681991;
   DATA[401,37] := 189.727;
   DATA[401,38] := 0.000128152;
   DATA[401,39] := 1.0;
   DATA[402,0] := 2.619543;
   DATA[402,1] := 527.7926;
   DATA[402,2] := 2.0;
   DATA[402,3] := 2.0;
   DATA[402,4] := 262.0802;
   DATA[402,5] := 8.393873;
   DATA[402,6] := 328.0441;
   DATA[402,7] := 2.441803;
   DATA[402,8] := 2.0;
   DATA[402,9] := 2.0;
   DATA[402,10] := 2.0;
   DATA[402,11] := 19.55311;
   DATA[402,12] := 2.209269;
   DATA[402,13] := 975.431;
   DATA[402,14] := 1.0;
   DATA[402,15] := 2.0;
   DATA[402,16] := 1.0;
   DATA[402,17] := 1.0;
   DATA[402,18] := 1.0;
   DATA[402,19] := 2.0;
   DATA[402,20] := 148.808;
   DATA[402,21] := 155.7293;
   DATA[402,22] := 1.715952;
   DATA[402,23] := 973.6734;
   DATA[402,24] := 2.0;
   DATA[402,25] := 2.0;
   DATA[402,26] := 7.879582;
   DATA[402,27] := 144.9628;
   DATA[402,28] := 263.7465;
   DATA[402,29] := 12.15073;
   DATA[402,30] := 1.729172;
   DATA[402,31] := 1.292174;
   DATA[402,32] := 0.736421;
   DATA[402,33] := 0.3066329;
   DATA[402,34] := 2.0;
   DATA[402,35] := 251.1055;
   DATA[402,36] := 1.681991;
   DATA[402,37] := 189.727;
   DATA[402,38] := 0.000128152;
   DATA[402,39] := 1.0;
   DATA[403,0] := 2.61538;
   DATA[403,1] := 527.6748;
   DATA[403,2] := 2.0;
   DATA[403,3] := 2.0;
   DATA[403,4] := 262.0802;
   DATA[403,5] := 8.393873;
   DATA[403,6] := 328.0441;
   DATA[403,7] := 2.441803;
   DATA[403,8] := 2.0;
   DATA[403,9] := 2.0;
   DATA[403,10] := 2.0;
   DATA[403,11] := 19.47948;
   DATA[403,12] := 2.209269;
   DATA[403,13] := 975.5912;
   DATA[403,14] := 1.0;
   DATA[403,15] := 2.0;
   DATA[403,16] := 1.0;
   DATA[403,17] := 1.0;
   DATA[403,18] := 1.0;
   DATA[403,19] := 2.0;
   DATA[403,20] := 148.808;
   DATA[403,21] := 155.7293;
   DATA[403,22] := 1.715567;
   DATA[403,23] := 974.0579;
   DATA[403,24] := 2.0;
   DATA[403,25] := 2.0;
   DATA[403,26] := 7.879582;
   DATA[403,27] := 144.9628;
   DATA[403,28] := 263.7465;
   DATA[403,29] := 12.15073;
   DATA[403,30] := 1.729172;
   DATA[403,31] := 1.282311;
   DATA[403,32] := 0.7357808;
   DATA[403,33] := 0.3066329;
   DATA[403,34] := 2.0;
   DATA[403,35] := 251.1055;
   DATA[403,36] := 1.681991;
   DATA[403,37] := 189.727;
   DATA[403,38] := 0.000128152;
   DATA[403,39] := 1.0;
   DATA[404,0] := 2.603209;
   DATA[404,1] := 528.3813;
   DATA[404,2] := 2.0;
   DATA[404,3] := 2.0;
   DATA[404,4] := 262.0802;
   DATA[404,5] := 8.393873;
   DATA[404,6] := 328.0441;
   DATA[404,7] := 2.441803;
   DATA[404,8] := 2.0;
   DATA[404,9] := 2.0;
   DATA[404,10] := 2.0;
   DATA[404,11] := 19.47948;
   DATA[404,12] := 2.209269;
   DATA[404,13] := 975.6713;
   DATA[404,14] := 1.0;
   DATA[404,15] := 2.0;
   DATA[404,16] := 1.0;
   DATA[404,17] := 1.0;
   DATA[404,18] := 1.0;
   DATA[404,19] := 2.0;
   DATA[404,20] := 148.808;
   DATA[404,21] := 155.7293;
   DATA[404,22] := 1.715567;
   DATA[404,23] := 974.2502;
   DATA[404,24] := 2.0;
   DATA[404,25] := 2.0;
   DATA[404,26] := 7.879582;
   DATA[404,27] := 145.0397;
   DATA[404,28] := 263.4261;
   DATA[404,29] := 12.15073;
   DATA[404,30] := 1.729172;
   DATA[404,31] := 1.265147;
   DATA[404,32] := 0.7357808;
   DATA[404,33] := 0.3066329;
   DATA[404,34] := 2.0;
   DATA[404,35] := 251.1055;
   DATA[404,36] := 1.617916;
   DATA[404,37] := 189.727;
   DATA[404,38] := 0.000128152;
   DATA[404,39] := 1.0;
   DATA[405,0] := 2.583992;
   DATA[405,1] := 528.7347;
   DATA[405,2] := 2.0;
   DATA[405,3] := 2.0;
   DATA[405,4] := 262.0802;
   DATA[405,5] := 8.393873;
   DATA[405,6] := 328.0441;
   DATA[405,7] := 2.440778;
   DATA[405,8] := 2.0;
   DATA[405,9] := 2.0;
   DATA[405,10] := 2.0;
   DATA[405,11] := 19.51149;
   DATA[405,12] := 2.209013;
   DATA[405,13] := 975.8315;
   DATA[405,14] := 1.0;
   DATA[405,15] := 2.0;
   DATA[405,16] := 1.0;
   DATA[405,17] := 1.0;
   DATA[405,18] := 1.0;
   DATA[405,19] := 2.0;
   DATA[405,20] := 148.808;
   DATA[405,21] := 155.7293;
   DATA[405,22] := 1.717489;
   DATA[405,23] := 974.4809;
   DATA[405,24] := 2.0;
   DATA[405,25] := 2.0;
   DATA[405,26] := 7.879582;
   DATA[405,27] := 145.0397;
   DATA[405,28] := 263.4261;
   DATA[405,29] := 12.15073;
   DATA[405,30] := 1.729172;
   DATA[405,31] := 1.26694;
   DATA[405,32] := 0.7357808;
   DATA[405,33] := 0.3066329;
   DATA[405,34] := 2.0;
   DATA[405,35] := 251.1055;
   DATA[405,36] := 1.617916;
   DATA[405,37] := 189.727;
   DATA[405,38] := 0.000128152;
   DATA[405,39] := 1.0;
   DATA[406,0] := 2.568299;
   DATA[406,1] := 529.0486;
   DATA[406,2] := 2.0;
   DATA[406,3] := 2.0;
   DATA[406,4] := 262.0802;
   DATA[406,5] := 8.393873;
   DATA[406,6] := 328.0441;
   DATA[406,7] := 2.440265;
   DATA[406,8] := 2.0;
   DATA[406,9] := 2.0;
   DATA[406,10] := 2.0;
   DATA[406,11] := 19.57232;
   DATA[406,12] := 2.208628;
   DATA[406,13] := 975.9517;
   DATA[406,14] := 1.0;
   DATA[406,15] := 2.0;
   DATA[406,16] := 1.0;
   DATA[406,17] := 1.0;
   DATA[406,18] := 1.0;
   DATA[406,19] := 2.0;
   DATA[406,20] := 148.808;
   DATA[406,21] := 155.7293;
   DATA[406,22] := 1.717489;
   DATA[406,23] := 975.2499;
   DATA[406,24] := 2.0;
   DATA[406,25] := 2.0;
   DATA[406,26] := 7.879582;
   DATA[406,27] := 145.0397;
   DATA[406,28] := 263.4261;
   DATA[406,29] := 11.95847;
   DATA[406,30] := 1.729172;
   DATA[406,31] := 1.272576;
   DATA[406,32] := 0.7357808;
   DATA[406,33] := 0.3066329;
   DATA[406,34] := 2.0;
   DATA[406,35] := 251.1055;
   DATA[406,36] := 1.617916;
   DATA[406,37] := 189.727;
   DATA[406,38] := 0.000128152;
   DATA[406,39] := 1.0;
   DATA[407,0] := 2.54588;
   DATA[407,1] := 529.9122;
   DATA[407,2] := 2.0;
   DATA[407,3] := 2.0;
   DATA[407,4] := 262.0802;
   DATA[407,5] := 8.393873;
   DATA[407,6] := 328.0441;
   DATA[407,7] := 2.439753;
   DATA[407,8] := 2.0;
   DATA[407,9] := 2.0;
   DATA[407,10] := 2.0;
   DATA[407,11] := 19.62354;
   DATA[407,12] := 2.208628;
   DATA[407,13] := 976.192;
   DATA[407,14] := 1.0;
   DATA[407,15] := 2.0;
   DATA[407,16] := 1.0;
   DATA[407,17] := 1.0;
   DATA[407,18] := 1.0;
   DATA[407,19] := 2.0;
   DATA[407,20] := 148.808;
   DATA[407,21] := 155.7293;
   DATA[407,22] := 1.717489;
   DATA[407,23] := 975.7498;
   DATA[407,24] := 2.0;
   DATA[407,25] := 2.0;
   DATA[407,26] := 7.879582;
   DATA[407,27] := 145.0397;
   DATA[407,28] := 263.5863;
   DATA[407,29] := 11.88157;
   DATA[407,30] := 1.726737;
   DATA[407,31] := 1.281542;
   DATA[407,32] := 0.7357808;
   DATA[407,33] := 0.3066329;
   DATA[407,34] := 2.0;
   DATA[407,35] := 250.9933;
   DATA[407,36] := 1.617916;
   DATA[407,37] := 189.727;
   DATA[407,38] := 0.000128152;
   DATA[407,39] := 1.0;
   DATA[408,0] := 2.531147;
   DATA[408,1] := 531.0113;
   DATA[408,2] := 2.0;
   DATA[408,3] := 2.0;
   DATA[408,4] := 262.0802;
   DATA[408,5] := 8.393553;
   DATA[408,6] := 328.0441;
   DATA[408,7] := 2.439496;
   DATA[408,8] := 2.0;
   DATA[408,9] := 2.0;
   DATA[408,10] := 2.0;
   DATA[408,11] := 19.62674;
   DATA[408,12] := 2.209397;
   DATA[408,13] := 976.152;
   DATA[408,14] := 1.0;
   DATA[408,15] := 2.0;
   DATA[408,16] := 1.0;
   DATA[408,17] := 1.0;
   DATA[408,18] := 1.0;
   DATA[408,19] := 2.0;
   DATA[408,20] := 148.808;
   DATA[408,21] := 155.7293;
   DATA[408,22] := 1.717489;
   DATA[408,23] := 976.2112;
   DATA[408,24] := 2.0;
   DATA[408,25] := 2.0;
   DATA[408,26] := 7.879582;
   DATA[408,27] := 145.0397;
   DATA[408,28] := 263.5863;
   DATA[408,29] := 11.88157;
   DATA[408,30] := 1.726352;
   DATA[408,31] := 1.282439;
   DATA[408,32] := 0.7357808;
   DATA[408,33] := 0.3066329;
   DATA[408,34] := 2.0;
   DATA[408,35] := 250.9132;
   DATA[408,36] := 1.730048;
   DATA[408,37] := 189.727;
   DATA[408,38] := 0.000128152;
   DATA[408,39] := 1.0;
   DATA[409,0] := 2.512891;
   DATA[409,1] := 531.6786;
   DATA[409,2] := 2.0;
   DATA[409,3] := 2.0;
   DATA[409,4] := 262.0802;
   DATA[409,5] := 8.393553;
   DATA[409,6] := 328.0441;
   DATA[409,7] := 2.439496;
   DATA[409,8] := 2.0;
   DATA[409,9] := 2.0;
   DATA[409,10] := 2.0;
   DATA[409,11] := 19.69396;
   DATA[409,12] := 2.21119;
   DATA[409,13] := 975.8716;
   DATA[409,14] := 1.0;
   DATA[409,15] := 2.0;
   DATA[409,16] := 1.0;
   DATA[409,17] := 1.0;
   DATA[409,18] := 1.0;
   DATA[409,19] := 2.0;
   DATA[409,20] := 148.808;
   DATA[409,21] := 155.7293;
   DATA[409,22] := 1.717489;
   DATA[409,23] := 976.7111;
   DATA[409,24] := 2.0;
   DATA[409,25] := 2.0;
   DATA[409,26] := 7.879582;
   DATA[409,27] := 145.0397;
   DATA[409,28] := 263.5863;
   DATA[409,29] := 12.22763;
   DATA[409,30] := 1.725327;
   DATA[409,31] := 1.282439;
   DATA[409,32] := 0.7357808;
   DATA[409,33] := 0.3066329;
   DATA[409,34] := 2.0;
   DATA[409,35] := 250.9132;
   DATA[409,36] := 1.730048;
   DATA[409,37] := 189.727;
   DATA[409,38] := 0.000128152;
   DATA[409,39] := 1.0;
   DATA[410,0] := 2.50008;
   DATA[410,1] := 532.1889;
   DATA[410,2] := 2.0;
   DATA[410,3] := 2.0;
   DATA[410,4] := 262.0802;
   DATA[410,5] := 8.39163;
   DATA[410,6] := 328.0441;
   DATA[410,7] := 2.439496;
   DATA[410,8] := 2.0;
   DATA[410,9] := 2.0;
   DATA[410,10] := 2.0;
   DATA[410,11] := 19.70677;
   DATA[410,12] := 2.21119;
   DATA[410,13] := 975.9517;
   DATA[410,14] := 1.0;
   DATA[410,15] := 2.0;
   DATA[410,16] := 1.0;
   DATA[410,17] := 1.0;
   DATA[410,18] := 1.0;
   DATA[410,19] := 2.0;
   DATA[410,20] := 148.808;
   DATA[410,21] := 155.7293;
   DATA[410,22] := 1.717489;
   DATA[410,23] := 976.6727;
   DATA[410,24] := 2.0;
   DATA[410,25] := 2.0;
   DATA[410,26] := 7.87766;
   DATA[410,27] := 145.0397;
   DATA[410,28] := 263.5863;
   DATA[410,29] := 12.22763;
   DATA[410,30] := 1.725327;
   DATA[410,31] := 1.294095;
   DATA[410,32] := 0.7357808;
   DATA[410,33] := 0.3066329;
   DATA[410,34] := 2.0;
   DATA[410,35] := 250.9132;
   DATA[410,36] := 1.730048;
   DATA[410,37] := 189.727;
   DATA[410,38] := 0.000128152;
   DATA[410,39] := 1.0;
   DATA[411,0] := 2.486308;
   DATA[411,1] := 532.5814;
   DATA[411,2] := 2.0;
   DATA[411,3] := 2.0;
   DATA[411,4] := 262.0802;
   DATA[411,5] := 8.39163;
   DATA[411,6] := 328.0441;
   DATA[411,7] := 2.441034;
   DATA[411,8] := 2.0;
   DATA[411,9] := 2.0;
   DATA[411,10] := 2.0;
   DATA[411,11] := 19.70677;
   DATA[411,12] := 2.21119;
   DATA[411,13] := 975.7915;
   DATA[411,14] := 1.0;
   DATA[411,15] := 2.0;
   DATA[411,16] := 1.0;
   DATA[411,17] := 1.0;
   DATA[411,18] := 1.0;
   DATA[411,19] := 2.0;
   DATA[411,20] := 148.808;
   DATA[411,21] := 155.7293;
   DATA[411,22] := 1.717489;
   DATA[411,23] := 976.9034;
   DATA[411,24] := 2.0;
   DATA[411,25] := 2.0;
   DATA[411,26] := 7.87766;
   DATA[411,27] := 145.0397;
   DATA[411,28] := 263.5863;
   DATA[411,29] := 12.22763;
   DATA[411,30] := 1.725327;
   DATA[411,31] := 1.297041;
   DATA[411,32] := 0.7355248;
   DATA[411,33] := 0.3066329;
   DATA[411,34] := 2.0;
   DATA[411,35] := 250.9132;
   DATA[411,36] := 1.69801;
   DATA[411,37] := 189.727;
   DATA[411,38] := 0.000128152;
   DATA[411,39] := 1.0;
   DATA[412,0] := 2.471896;
   DATA[412,1] := 532.7384;
   DATA[412,2] := 2.0;
   DATA[412,3] := 2.0;
   DATA[412,4] := 262.0802;
   DATA[412,5] := 8.39163;
   DATA[412,6] := 328.0441;
   DATA[412,7] := 2.441034;
   DATA[412,8] := 2.0;
   DATA[412,9] := 2.0;
   DATA[412,10] := 2.0;
   DATA[412,11] := 19.70677;
   DATA[412,12] := 2.210934;
   DATA[412,13] := 975.9517;
   DATA[412,14] := 1.0;
   DATA[412,15] := 2.0;
   DATA[412,16] := 1.0;
   DATA[412,17] := 1.0;
   DATA[412,18] := 1.0;
   DATA[412,19] := 2.0;
   DATA[412,20] := 148.808;
   DATA[412,21] := 155.7806;
   DATA[412,22] := 1.717489;
   DATA[412,23] := 976.5573;
   DATA[412,24] := 2.0;
   DATA[412,25] := 2.0;
   DATA[412,26] := 7.87766;
   DATA[412,27] := 145.0397;
   DATA[412,28] := 263.5863;
   DATA[412,29] := 11.92002;
   DATA[412,30] := 1.725327;
   DATA[412,31] := 1.291533;
   DATA[412,32] := 0.7351407;
   DATA[412,33] := 0.3066329;
   DATA[412,34] := 2.0;
   DATA[412,35] := 250.9132;
   DATA[412,36] := 1.617916;
   DATA[412,37] := 189.727;
   DATA[412,38] := 0.000128152;
   DATA[412,39] := 1.0;
   DATA[413,0] := 2.460045;
   DATA[413,1] := 532.3459;
   DATA[413,2] := 2.0;
   DATA[413,3] := 2.0;
   DATA[413,4] := 262.0802;
   DATA[413,5] := 8.39163;
   DATA[413,6] := 328.0441;
   DATA[413,7] := 2.441034;
   DATA[413,8] := 2.0;
   DATA[413,9] := 2.0;
   DATA[413,10] := 2.0;
   DATA[413,11] := 19.70677;
   DATA[413,12] := 2.210934;
   DATA[413,13] := 975.8315;
   DATA[413,14] := 1.0;
   DATA[413,15] := 2.0;
   DATA[413,16] := 1.0;
   DATA[413,17] := 1.0;
   DATA[413,18] := 1.0;
   DATA[413,19] := 2.0;
   DATA[413,20] := 148.808;
   DATA[413,21] := 155.7806;
   DATA[413,22] := 1.717489;
   DATA[413,23] := 977.0956;
   DATA[413,24] := 2.0;
   DATA[413,25] := 2.0;
   DATA[413,26] := 7.87766;
   DATA[413,27] := 145.0397;
   DATA[413,28] := 263.5863;
   DATA[413,29] := 11.92002;
   DATA[413,30] := 1.725327;
   DATA[413,31] := 1.281798;
   DATA[413,32] := 0.7351407;
   DATA[413,33] := 0.3081703;
   DATA[413,34] := 2.0;
   DATA[413,35] := 250.9132;
   DATA[413,36] := 1.617916;
   DATA[413,37] := 189.727;
   DATA[413,38] := 0.000128152;
   DATA[413,39] := 1.0;
   DATA[414,0] := 2.443391;
   DATA[414,1] := 532.1889;
   DATA[414,2] := 2.0;
   DATA[414,3] := 2.0;
   DATA[414,4] := 262.0802;
   DATA[414,5] := 8.39163;
   DATA[414,6] := 328.0441;
   DATA[414,7] := 2.440521;
   DATA[414,8] := 2.0;
   DATA[414,9] := 2.0;
   DATA[414,10] := 2.0;
   DATA[414,11] := 19.70677;
   DATA[414,12] := 2.210934;
   DATA[414,13] := 975.7915;
   DATA[414,14] := 1.0;
   DATA[414,15] := 2.0;
   DATA[414,16] := 1.0;
   DATA[414,17] := 1.0;
   DATA[414,18] := 1.0;
   DATA[414,19] := 2.0;
   DATA[414,20] := 148.808;
   DATA[414,21] := 155.7806;
   DATA[414,22] := 1.717489;
   DATA[414,23] := 976.9803;
   DATA[414,24] := 2.0;
   DATA[414,25] := 2.0;
   DATA[414,26] := 7.87766;
   DATA[414,27] := 145.0397;
   DATA[414,28] := 263.5863;
   DATA[414,29] := 11.92002;
   DATA[414,30] := 1.725327;
   DATA[414,31] := 1.273216;
   DATA[414,32] := 0.7351407;
   DATA[414,33] := 0.3081703;
   DATA[414,34] := 2.0;
   DATA[414,35] := 250.9132;
   DATA[414,36] := 1.617916;
   DATA[414,37] := 189.727;
   DATA[414,38] := 0.000128152;
   DATA[414,39] := 1.0;
   DATA[415,0] := 2.434423;
   DATA[415,1] := 531.8749;
   DATA[415,2] := 2.0;
   DATA[415,3] := 2.0;
   DATA[415,4] := 262.0802;
   DATA[415,5] := 8.391951;
   DATA[415,6] := 328.0441;
   DATA[415,7] := 2.440521;
   DATA[415,8] := 2.0;
   DATA[415,9] := 2.0;
   DATA[415,10] := 2.0;
   DATA[415,11] := 19.76759;
   DATA[415,12] := 2.210934;
   DATA[415,13] := 975.5912;
   DATA[415,14] := 1.0;
   DATA[415,15] := 2.0;
   DATA[415,16] := 1.0;
   DATA[415,17] := 1.0;
   DATA[415,18] := 1.0;
   DATA[415,19] := 2.0;
   DATA[415,20] := 148.808;
   DATA[415,21] := 155.7806;
   DATA[415,22] := 1.717489;
   DATA[415,23] := 977.5186;
   DATA[415,24] := 2.0;
   DATA[415,25] := 2.0;
   DATA[415,26] := 7.87766;
   DATA[415,27] := 145.0397;
   DATA[415,28] := 263.5863;
   DATA[415,29] := 11.92002;
   DATA[415,30] := 1.725327;
   DATA[415,31] := 1.271551;
   DATA[415,32] := 0.7351407;
   DATA[415,33] := 0.3081703;
   DATA[415,34] := 2.0;
   DATA[415,35] := 250.9132;
   DATA[415,36] := 1.617916;
   DATA[415,37] := 189.727;
   DATA[415,38] := 0.000128152;
   DATA[415,39] := 1.0;
   DATA[416,0] := 2.426416;
   DATA[416,1] := 531.1291;
   DATA[416,2] := 2.0;
   DATA[416,3] := 2.0;
   DATA[416,4] := 262.0802;
   DATA[416,5] := 8.393232;
   DATA[416,6] := 328.0441;
   DATA[416,7] := 2.439625;
   DATA[416,8] := 2.0;
   DATA[416,9] := 2.0;
   DATA[416,10] := 2.0;
   DATA[416,11] := 19.7804;
   DATA[416,12] := 2.21055;
   DATA[416,13] := 975.6313;
   DATA[416,14] := 1.0;
   DATA[416,15] := 2.0;
   DATA[416,16] := 1.0;
   DATA[416,17] := 1.0;
   DATA[416,18] := 1.0;
   DATA[416,19] := 2.0;
   DATA[416,20] := 148.808;
   DATA[416,21] := 155.7806;
   DATA[416,22] := 1.717489;
   DATA[416,23] := 977.557;
   DATA[416,24] := 2.0;
   DATA[416,25] := 2.0;
   DATA[416,26] := 7.87766;
   DATA[416,27] := 145.0397;
   DATA[416,28] := 263.5863;
   DATA[416,29] := 11.92002;
   DATA[416,30] := 1.725327;
   DATA[416,31] := 1.275906;
   DATA[416,32] := 0.7351407;
   DATA[416,33] := 0.3083624;
   DATA[416,34] := 2.0;
   DATA[416,35] := 250.9132;
   DATA[416,36] := 1.617916;
   DATA[416,37] := 189.5347;
   DATA[416,38] := 0.000128152;
   DATA[416,39] := 1.0;
   DATA[417,0] := 2.422253;
   DATA[417,1] := 530.4225;
   DATA[417,2] := 2.0;
   DATA[417,3] := 2.0;
   DATA[417,4] := 262.0802;
   DATA[417,5] := 8.393553;
   DATA[417,6] := 328.0441;
   DATA[417,7] := 2.43924;
   DATA[417,8] := 2.0;
   DATA[417,9] := 2.0;
   DATA[417,10] := 2.0;
   DATA[417,11] := 19.7804;
   DATA[417,12] := 2.210037;
   DATA[417,13] := 975.6713;
   DATA[417,14] := 1.0;
   DATA[417,15] := 2.0;
   DATA[417,16] := 1.0;
   DATA[417,17] := 1.0;
   DATA[417,18] := 1.0;
   DATA[417,19] := 2.0;
   DATA[417,20] := 148.808;
   DATA[417,21] := 155.7806;
   DATA[417,22] := 1.717489;
   DATA[417,23] := 977.4417;
   DATA[417,24] := 2.0;
   DATA[417,25] := 2.0;
   DATA[417,26] := 7.87766;
   DATA[417,27] := 145.0397;
   DATA[417,28] := 263.5863;
   DATA[417,29] := 12.15073;
   DATA[417,30] := 1.72789;
   DATA[417,31] := 1.290893;
   DATA[417,32] := 0.7351407;
   DATA[417,33] := 0.3083624;
   DATA[417,34] := 2.0;
   DATA[417,35] := 250.9132;
   DATA[417,36] := 1.617916;
   DATA[417,37] := 189.5347;
   DATA[417,38] := 0.000128152;
   DATA[417,39] := 1.0;
   DATA[418,0] := 2.428018;
   DATA[418,1] := 530.1085;
   DATA[418,2] := 2.0;
   DATA[418,3] := 2.0;
   DATA[418,4] := 262.0802;
   DATA[418,5] := 8.393553;
   DATA[418,6] := 328.0441;
   DATA[418,7] := 2.43924;
   DATA[418,8] := 2.0;
   DATA[418,9] := 2.0;
   DATA[418,10] := 2.0;
   DATA[418,11] := 19.72598;
   DATA[418,12] := 2.210037;
   DATA[418,13] := 975.3509;
   DATA[418,14] := 1.0;
   DATA[418,15] := 2.0;
   DATA[418,16] := 1.0;
   DATA[418,17] := 1.0;
   DATA[418,18] := 1.0;
   DATA[418,19] := 2.0;
   DATA[418,20] := 148.808;
   DATA[418,21] := 155.7806;
   DATA[418,22] := 1.717489;
   DATA[418,23] := 977.3648;
   DATA[418,24] := 2.0;
   DATA[418,25] := 2.0;
   DATA[418,26] := 7.87766;
   DATA[418,27] := 145.0397;
   DATA[418,28] := 263.5863;
   DATA[418,29] := 12.41989;
   DATA[418,30] := 1.72789;
   DATA[418,31] := 1.291918;
   DATA[418,32] := 0.7351407;
   DATA[418,33] := 0.3083624;
   DATA[418,34] := 2.0;
   DATA[418,35] := 250.9132;
   DATA[418,36] := 1.617916;
   DATA[418,37] := 189.5347;
   DATA[418,38] := 0.000128152;
   DATA[418,39] := 1.0;
   DATA[419,0] := 2.468052;
   DATA[419,1] := 529.7159;
   DATA[419,2] := 2.0;
   DATA[419,3] := 2.0;
   DATA[419,4] := 262.0802;
   DATA[419,5] := 8.393553;
   DATA[419,6] := 328.0441;
   DATA[419,7] := 2.43924;
   DATA[419,8] := 2.0;
   DATA[419,9] := 2.0;
   DATA[419,10] := 2.0;
   DATA[419,11] := 19.72598;
   DATA[419,12] := 2.209909;
   DATA[419,13] := 975.5912;
   DATA[419,14] := 1.0;
   DATA[419,15] := 2.0;
   DATA[419,16] := 1.0;
   DATA[419,17] := 1.0;
   DATA[419,18] := 1.0;
   DATA[419,19] := 2.0;
   DATA[419,20] := 148.808;
   DATA[419,21] := 155.7806;
   DATA[419,22] := 1.717489;
   DATA[419,23] := 977.3264;
   DATA[419,24] := 2.0;
   DATA[419,25] := 2.0;
   DATA[419,26] := 7.87766;
   DATA[419,27] := 145.0397;
   DATA[419,28] := 263.5863;
   DATA[419,29] := 12.41989;
   DATA[419,30] := 1.72789;
   DATA[419,31] := 1.301652;
   DATA[419,32] := 0.7351407;
   DATA[419,33] := 0.3083624;
   DATA[419,34] := 2.0;
   DATA[419,35] := 250.9132;
   DATA[419,36] := 1.617916;
   DATA[419,37] := 189.6949;
   DATA[419,38] := 0.000128152;
   DATA[419,39] := 1.0;
   DATA[420,0] := 2.520257;
   DATA[420,1] := 529.7159;
   DATA[420,2] := 2.0;
   DATA[420,3] := 2.0;
   DATA[420,4] := 262.0802;
   DATA[420,5] := 8.393553;
   DATA[420,6] := 328.0441;
   DATA[420,7] := 2.439753;
   DATA[420,8] := 2.0;
   DATA[420,9] := 2.0;
   DATA[420,10] := 2.0;
   DATA[420,11] := 19.72598;
   DATA[420,12] := 2.209013;
   DATA[420,13] := 975.7915;
   DATA[420,14] := 1.0;
   DATA[420,15] := 2.0;
   DATA[420,16] := 1.0;
   DATA[420,17] := 1.0;
   DATA[420,18] := 1.0;
   DATA[420,19] := 2.0;
   DATA[420,20] := 148.808;
   DATA[420,21] := 155.7806;
   DATA[420,22] := 1.717489;
   DATA[420,23] := 977.2879;
   DATA[420,24] := 2.0;
   DATA[420,25] := 2.0;
   DATA[420,26] := 7.87766;
   DATA[420,27] := 145.0397;
   DATA[420,28] := 263.5863;
   DATA[420,29] := 12.41989;
   DATA[420,30] := 1.72789;
   DATA[420,31] := 1.296401;
   DATA[420,32] := 0.7351407;
   DATA[420,33] := 0.3083624;
   DATA[420,34] := 2.0;
   DATA[420,35] := 250.9132;
   DATA[420,36] := 1.617916;
   DATA[420,37] := 189.727;
   DATA[420,38] := 0.000128152;
   DATA[420,39] := 1.0;
   DATA[421,0] := 2.559972;
   DATA[421,1] := 529.5982;
   DATA[421,2] := 2.0;
   DATA[421,3] := 2.0;
   DATA[421,4] := 262.2084;
   DATA[421,5] := 8.393553;
   DATA[421,6] := 328.2748;
   DATA[421,7] := 2.440393;
   DATA[421,8] := 2.0;
   DATA[421,9] := 2.0;
   DATA[421,10] := 2.0;
   DATA[421,11] := 19.65555;
   DATA[421,12] := 2.211831;
   DATA[421,13] := 975.7514;
   DATA[421,14] := 1.0;
   DATA[421,15] := 2.0;
   DATA[421,16] := 1.0;
   DATA[421,17] := 1.0;
   DATA[421,18] := 1.0;
   DATA[421,19] := 2.0;
   DATA[421,20] := 148.808;
   DATA[421,21] := 155.8062;
   DATA[421,22] := 1.717489;
   DATA[421,23] := 977.2879;
   DATA[421,24] := 2.0;
   DATA[421,25] := 2.0;
   DATA[421,26] := 7.87766;
   DATA[421,27] := 145.0397;
   DATA[421,28] := 263.5863;
   DATA[421,29] := 11.95847;
   DATA[421,30] := 1.72789;
   DATA[421,31] := 1.292046;
   DATA[421,32] := 0.7351407;
   DATA[421,33] := 0.3083624;
   DATA[421,34] := 2.0;
   DATA[421,35] := 250.9132;
   DATA[421,36] := 1.617916;
   DATA[421,37] := 189.727;
   DATA[421,38] := 0.000128152;
   DATA[421,39] := 1.0;
   DATA[422,0] := 2.603209;
   DATA[422,1] := 529.0486;
   DATA[422,2] := 2.0;
   DATA[422,3] := 2.0;
   DATA[422,4] := 262.2404;
   DATA[422,5] := 8.393553;
   DATA[422,6] := 328.2748;
   DATA[422,7] := 2.440778;
   DATA[422,8] := 2.0;
   DATA[422,9] := 2.0;
   DATA[422,10] := 2.0;
   DATA[422,11] := 19.65555;
   DATA[422,12] := 2.211831;
   DATA[422,13] := 975.5511;
   DATA[422,14] := 1.0;
   DATA[422,15] := 2.0;
   DATA[422,16] := 1.0;
   DATA[422,17] := 1.0;
   DATA[422,18] := 1.0;
   DATA[422,19] := 2.0;
   DATA[422,20] := 148.808;
   DATA[422,21] := 156.0625;
   DATA[422,22] := 1.717489;
   DATA[422,23] := 977.2879;
   DATA[422,24] := 2.0;
   DATA[422,25] := 2.0;
   DATA[422,26] := 7.87766;
   DATA[422,27] := 145.0397;
   DATA[422,28] := 263.5863;
   DATA[422,29] := 11.95847;
   DATA[422,30] := 1.7293;
   DATA[422,31] := 1.291405;
   DATA[422,32] := 0.7351407;
   DATA[422,33] := 0.3083624;
   DATA[422,34] := 2.0;
   DATA[422,35] := 250.9132;
   DATA[422,36] := 1.617916;
   DATA[422,37] := 189.727;
   DATA[422,38] := 0.000128152;
   DATA[422,39] := 1.0;
   DATA[423,0] := 2.632354;
   DATA[423,1] := 529.402;
   DATA[423,2] := 2.0;
   DATA[423,3] := 2.0;
   DATA[423,4] := 262.2404;
   DATA[423,5] := 8.393553;
   DATA[423,6] := 328.2748;
   DATA[423,7] := 2.441419;
   DATA[423,8] := 2.0;
   DATA[423,9] := 2.0;
   DATA[423,10] := 2.0;
   DATA[423,11] := 19.65555;
   DATA[423,12] := 2.211831;
   DATA[423,13] := 975.9918;
   DATA[423,14] := 1.0;
   DATA[423,15] := 2.0;
   DATA[423,16] := 1.0;
   DATA[423,17] := 1.0;
   DATA[423,18] := 1.0;
   DATA[423,19] := 2.0;
   DATA[423,20] := 148.808;
   DATA[423,21] := 156.0625;
   DATA[423,22] := 1.717489;
   DATA[423,23] := 977.3648;
   DATA[423,24] := 2.0;
   DATA[423,25] := 2.0;
   DATA[423,26] := 7.878621;
   DATA[423,27] := 145.0397;
   DATA[423,28] := 263.5863;
   DATA[423,29] := 11.95847;
   DATA[423,30] := 1.7293;
   DATA[423,31] := 1.291405;
   DATA[423,32] := 0.7351407;
   DATA[423,33] := 0.3083624;
   DATA[423,34] := 2.0;
   DATA[423,35] := 250.9132;
   DATA[423,36] := 1.617916;
   DATA[423,37] := 189.6629;
   DATA[423,38] := 0.000128152;
   DATA[423,39] := 1.0;
   DATA[424,0] := 2.649649;
   DATA[424,1] := 529.3627;
   DATA[424,2] := 2.0;
   DATA[424,3] := 2.0;
   DATA[424,4] := 262.2404;
   DATA[424,5] := 8.393553;
   DATA[424,6] := 327.9672;
   DATA[424,7] := 2.441419;
   DATA[424,8] := 2.0;
   DATA[424,9] := 2.0;
   DATA[424,10] := 2.0;
   DATA[424,11] := 19.66195;
   DATA[424,12] := 2.213624;
   DATA[424,13] := 976.4324;
   DATA[424,14] := 1.0;
   DATA[424,15] := 2.0;
   DATA[424,16] := 1.0;
   DATA[424,17] := 1.0;
   DATA[424,18] := 1.0;
   DATA[424,19] := 2.0;
   DATA[424,20] := 148.808;
   DATA[424,21] := 156.0625;
   DATA[424,22] := 1.717489;
   DATA[424,23] := 976.788;
   DATA[424,24] := 2.0;
   DATA[424,25] := 2.0;
   DATA[424,26] := 7.878621;
   DATA[424,27] := 145.0397;
   DATA[424,28] := 263.5863;
   DATA[424,29] := 11.95847;
   DATA[424,30] := 1.726737;
   DATA[424,31] := 1.291405;
   DATA[424,32] := 0.7351407;
   DATA[424,33] := 0.3083624;
   DATA[424,34] := 2.0;
   DATA[424,35] := 250.9132;
   DATA[424,36] := 1.617916;
   DATA[424,37] := 189.5347;
   DATA[424,38] := 0.000128152;
   DATA[424,39] := 1.0;
   DATA[425,0] := 2.66214;
   DATA[425,1] := 529.5982;
   DATA[425,2] := 2.0;
   DATA[425,3] := 2.0;
   DATA[425,4] := 262.2404;
   DATA[425,5] := 8.393553;
   DATA[425,6] := 327.9672;
   DATA[425,7] := 2.441419;
   DATA[425,8] := 2.0;
   DATA[425,9] := 2.0;
   DATA[425,10] := 2.0;
   DATA[425,11] := 19.66195;
   DATA[425,12] := 2.213624;
   DATA[425,13] := 976.4724;
   DATA[425,14] := 1.0;
   DATA[425,15] := 2.0;
   DATA[425,16] := 1.0;
   DATA[425,17] := 1.0;
   DATA[425,18] := 1.0;
   DATA[425,19] := 2.0;
   DATA[425,20] := 148.808;
   DATA[425,21] := 156.0625;
   DATA[425,22] := 1.717489;
   DATA[425,23] := 977.0956;
   DATA[425,24] := 2.0;
   DATA[425,25] := 2.0;
   DATA[425,26] := 7.878621;
   DATA[425,27] := 145.0397;
   DATA[425,28] := 263.5863;
   DATA[425,29] := 11.95847;
   DATA[425,30] := 1.726096;
   DATA[425,31] := 1.291405;
   DATA[425,32] := 0.7351407;
   DATA[425,33] := 0.3083624;
   DATA[425,34] := 2.0;
   DATA[425,35] := 250.9132;
   DATA[425,36] := 1.617916;
   DATA[425,37] := 189.5347;
   DATA[425,38] := 0.000128152;
   DATA[425,39] := 1.0;
   DATA[426,0] := 2.66214;
   DATA[426,1] := 529.5982;
   DATA[426,2] := 2.0;
   DATA[426,3] := 2.0;
   DATA[426,4] := 262.2404;
   DATA[426,5] := 8.393553;
   DATA[426,6] := 327.9672;
   DATA[426,7] := 2.441419;
   DATA[426,8] := 2.0;
   DATA[426,9] := 2.0;
   DATA[426,10] := 2.0;
   DATA[426,11] := 19.66195;
   DATA[426,12] := 2.213624;
   DATA[426,13] := 976.4724;
   DATA[426,14] := 1.0;
   DATA[426,15] := 2.0;
   DATA[426,16] := 1.0;
   DATA[426,17] := 1.0;
   DATA[426,18] := 1.0;
   DATA[426,19] := 2.0;
   DATA[426,20] := 148.808;
   DATA[426,21] := 156.0625;
   DATA[426,22] := 1.717489;
   DATA[426,23] := 977.0956;
   DATA[426,24] := 2.0;
   DATA[426,25] := 2.0;
   DATA[426,26] := 7.878621;
   DATA[426,27] := 145.0397;
   DATA[426,28] := 263.5863;
   DATA[426,29] := 11.95847;
   DATA[426,30] := 1.726096;
   DATA[426,31] := 1.291405;
   DATA[426,32] := 0.7351407;
   DATA[426,33] := 0.3083624;
   DATA[426,34] := 2.0;
   DATA[426,35] := 250.9132;
   DATA[426,36] := 1.617916;
   DATA[426,37] := 189.5347;
   DATA[426,38] := 0.000128152;
   DATA[426,39] := 1.0;
   DATA[427,0] := 2.66214;
   DATA[427,1] := 529.7159;
   DATA[427,2] := 2.0;
   DATA[427,3] := 2.0;
   DATA[427,4] := 262.2404;
   DATA[427,5] := 8.393553;
   DATA[427,6] := 327.9672;
   DATA[427,7] := 2.441419;
   DATA[427,8] := 2.0;
   DATA[427,9] := 2.0;
   DATA[427,10] := 2.0;
   DATA[427,11] := 19.66195;
   DATA[427,12] := 2.213624;
   DATA[427,13] := 976.3522;
   DATA[427,14] := 1.0;
   DATA[427,15] := 2.0;
   DATA[427,16] := 1.0;
   DATA[427,17] := 1.0;
   DATA[427,18] := 1.0;
   DATA[427,19] := 2.0;
   DATA[427,20] := 148.808;
   DATA[427,21] := 156.0625;
   DATA[427,22] := 1.717489;
   DATA[427,23] := 976.9803;
   DATA[427,24] := 2.0;
   DATA[427,25] := 2.0;
   DATA[427,26] := 7.878621;
   DATA[427,27] := 145.0397;
   DATA[427,28] := 263.5863;
   DATA[427,29] := 11.95847;
   DATA[427,30] := 1.726096;
   DATA[427,31] := 1.283464;
   DATA[427,32] := 0.7351407;
   DATA[427,33] := 0.3083624;
   DATA[427,34] := 2.0;
   DATA[427,35] := 250.9132;
   DATA[427,36] := 1.617916;
   DATA[427,37] := 189.5347;
   DATA[427,38] := 0.000128152;
   DATA[427,39] := 1.0;
   DATA[428,0] := 2.641002;
   DATA[428,1] := 529.5982;
   DATA[428,2] := 2.0;
   DATA[428,3] := 2.0;
   DATA[428,4] := 262.2404;
   DATA[428,5] := 8.393553;
   DATA[428,6] := 327.9672;
   DATA[428,7] := 2.441419;
   DATA[428,8] := 2.0;
   DATA[428,9] := 2.0;
   DATA[428,10] := 2.0;
   DATA[428,11] := 19.66195;
   DATA[428,12] := 2.213624;
   DATA[428,13] := 976.4724;
   DATA[428,14] := 1.0;
   DATA[428,15] := 2.0;
   DATA[428,16] := 1.0;
   DATA[428,17] := 1.0;
   DATA[428,18] := 1.0;
   DATA[428,19] := 2.0;
   DATA[428,20] := 148.808;
   DATA[428,21] := 156.0625;
   DATA[428,22] := 1.717489;
   DATA[428,23] := 976.9418;
   DATA[428,24] := 2.0;
   DATA[428,25] := 2.0;
   DATA[428,26] := 7.878621;
   DATA[428,27] := 145.1679;
   DATA[428,28] := 263.5863;
   DATA[428,29] := 11.95847;
   DATA[428,30] := 1.726096;
   DATA[428,31] := 1.281542;
   DATA[428,32] := 0.7351407;
   DATA[428,33] := 0.3083624;
   DATA[428,34] := 2.0;
   DATA[428,35] := 250.9132;
   DATA[428,36] := 1.617916;
   DATA[428,37] := 189.5347;
   DATA[428,38] := 0.000128152;
   DATA[428,39] := 1.0;
   DATA[429,0] := 2.629152;
   DATA[429,1] := 529.402;
   DATA[429,2] := 2.0;
   DATA[429,3] := 2.0;
   DATA[429,4] := 262.2404;
   DATA[429,5] := 8.393553;
   DATA[429,6] := 327.9672;
   DATA[429,7] := 2.441419;
   DATA[429,8] := 2.0;
   DATA[429,9] := 2.0;
   DATA[429,10] := 2.0;
   DATA[429,11] := 19.72277;
   DATA[429,12] := 2.213624;
   DATA[429,13] := 976.192;
   DATA[429,14] := 1.0;
   DATA[429,15] := 2.0;
   DATA[429,16] := 1.0;
   DATA[429,17] := 1.0;
   DATA[429,18] := 1.0;
   DATA[429,19] := 2.0;
   DATA[429,20] := 148.808;
   DATA[429,21] := 155.96;
   DATA[429,22] := 1.717489;
   DATA[429,23] := 977.2879;
   DATA[429,24] := 2.0;
   DATA[429,25] := 2.0;
   DATA[429,26] := 7.878621;
   DATA[429,27] := 145.1679;
   DATA[429,28] := 263.5863;
   DATA[429,29] := 11.95847;
   DATA[429,30] := 1.726096;
   DATA[429,31] := 1.288075;
   DATA[429,32] := 0.7351407;
   DATA[429,33] := 0.3083624;
   DATA[429,34] := 2.0;
   DATA[429,35] := 250.9132;
   DATA[429,36] := 1.617916;
   DATA[429,37] := 189.727;
   DATA[429,38] := 0.000128152;
   DATA[429,39] := 1.0;
   DATA[430,0] := 2.62723;
   DATA[430,1] := 529.402;
   DATA[430,2] := 2.0;
   DATA[430,3] := 2.0;
   DATA[430,4] := 262.2404;
   DATA[430,5] := 8.393553;
   DATA[430,6] := 327.9672;
   DATA[430,7] := 2.441419;
   DATA[430,8] := 2.0;
   DATA[430,9] := 2.0;
   DATA[430,10] := 2.0;
   DATA[430,11] := 19.73238;
   DATA[430,12] := 2.213624;
   DATA[430,13] := 976.0718;
   DATA[430,14] := 1.0;
   DATA[430,15] := 2.0;
   DATA[430,16] := 1.0;
   DATA[430,17] := 1.0;
   DATA[430,18] := 1.0;
   DATA[430,19] := 2.0;
   DATA[430,20] := 148.808;
   DATA[430,21] := 155.96;
   DATA[430,22] := 1.717489;
   DATA[430,23] := 977.0572;
   DATA[430,24] := 2.0;
   DATA[430,25] := 2.0;
   DATA[430,26] := 7.878621;
   DATA[430,27] := 145.1679;
   DATA[430,28] := 263.5863;
   DATA[430,29] := 11.95847;
   DATA[430,30] := 1.726096;
   DATA[430,31] := 1.285641;
   DATA[430,32] := 0.7360369;
   DATA[430,33] := 0.3083624;
   DATA[430,34] := 2.0;
   DATA[430,35] := 250.8652;
   DATA[430,36] := 1.617916;
   DATA[430,37] := 189.727;
   DATA[430,38] := 0.000128152;
   DATA[430,39] := 1.0;
   DATA[431,0] := 2.610896;
   DATA[431,1] := 529.8337;
   DATA[431,2] := 2.0;
   DATA[431,3] := 2.0;
   DATA[431,4] := 262.2404;
   DATA[431,5] := 8.393553;
   DATA[431,6] := 327.9672;
   DATA[431,7] := 2.441419;
   DATA[431,8] := 2.0;
   DATA[431,9] := 2.0;
   DATA[431,10] := 2.0;
   DATA[431,11] := 19.73238;
   DATA[431,12] := 2.213624;
   DATA[431,13] := 976.0318;
   DATA[431,14] := 1.0;
   DATA[431,15] := 2.0;
   DATA[431,16] := 1.0;
   DATA[431,17] := 1.0;
   DATA[431,18] := 1.0;
   DATA[431,19] := 2.0;
   DATA[431,20] := 148.808;
   DATA[431,21] := 155.96;
   DATA[431,22] := 1.717489;
   DATA[431,23] := 977.2879;
   DATA[431,24] := 2.0;
   DATA[431,25] := 2.0;
   DATA[431,26] := 7.878621;
   DATA[431,27] := 145.1679;
   DATA[431,28] := 263.5863;
   DATA[431,29] := 11.95847;
   DATA[431,30] := 1.728019;
   DATA[431,31] := 1.289484;
   DATA[431,32] := 0.7360369;
   DATA[431,33] := 0.3083624;
   DATA[431,34] := 2.0;
   DATA[431,35] := 250.8652;
   DATA[431,36] := 1.617916;
   DATA[431,37] := 189.727;
   DATA[431,38] := 0.000128152;
   DATA[431,39] := 1.0;
   DATA[432,0] := 2.588476;
   DATA[432,1] := 530.344;
   DATA[432,2] := 2.0;
   DATA[432,3] := 2.0;
   DATA[432,4] := 261.9841;
   DATA[432,5] := 8.393553;
   DATA[432,6] := 327.9672;
   DATA[432,7] := 2.439753;
   DATA[432,8] := 2.0;
   DATA[432,9] := 2.0;
   DATA[432,10] := 2.0;
   DATA[432,11] := 19.73238;
   DATA[432,12] := 2.213624;
   DATA[432,13] := 976.6727;
   DATA[432,14] := 1.0;
   DATA[432,15] := 2.0;
   DATA[432,16] := 1.0;
   DATA[432,17] := 1.0;
   DATA[432,18] := 1.0;
   DATA[432,19] := 2.0;
   DATA[432,20] := 148.808;
   DATA[432,21] := 155.96;
   DATA[432,22] := 1.717489;
   DATA[432,23] := 977.2879;
   DATA[432,24] := 2.0;
   DATA[432,25] := 2.0;
   DATA[432,26] := 7.878621;
   DATA[432,27] := 145.1679;
   DATA[432,28] := 263.5863;
   DATA[432,29] := 11.95847;
   DATA[432,30] := 1.728916;
   DATA[432,31] := 1.292686;
   DATA[432,32] := 0.7360369;
   DATA[432,33] := 0.3083624;
   DATA[432,34] := 2.0;
   DATA[432,35] := 250.8652;
   DATA[432,36] := 1.617916;
   DATA[432,37] := 189.727;
   DATA[432,38] := 0.000128152;
   DATA[432,39] := 1.0;
   DATA[433,0] := 2.567979;
   DATA[433,1] := 530.2263;
   DATA[433,2] := 2.0;
   DATA[433,3] := 2.0;
   DATA[433,4] := 261.9841;
   DATA[433,5] := 8.393553;
   DATA[433,6] := 327.9672;
   DATA[433,7] := 2.439753;
   DATA[433,8] := 2.0;
   DATA[433,9] := 2.0;
   DATA[433,10] := 2.0;
   DATA[433,11] := 19.70357;
   DATA[433,12] := 2.213624;
   DATA[433,13] := 976.7528;
   DATA[433,14] := 1.0;
   DATA[433,15] := 2.0;
   DATA[433,16] := 1.0;
   DATA[433,17] := 1.0;
   DATA[433,18] := 1.0;
   DATA[433,19] := 2.0;
   DATA[433,20] := 148.808;
   DATA[433,21] := 155.96;
   DATA[433,22] := 1.717489;
   DATA[433,23] := 977.557;
   DATA[433,24] := 2.0;
   DATA[433,25] := 2.0;
   DATA[433,26] := 7.878621;
   DATA[433,27] := 145.1679;
   DATA[433,28] := 263.5863;
   DATA[433,29] := 12.15073;
   DATA[433,30] := 1.728916;
   DATA[433,31] := 1.286153;
   DATA[433,32] := 0.7353967;
   DATA[433,33] := 0.3083624;
   DATA[433,34] := 2.0;
   DATA[433,35] := 250.8652;
   DATA[433,36] := 1.617916;
   DATA[433,37] := 189.727;
   DATA[433,38] := 0.000128152;
   DATA[433,39] := 1.0;
   DATA[434,0] := 2.553886;
   DATA[434,1] := 529.559;
   DATA[434,2] := 2.0;
   DATA[434,3] := 2.0;
   DATA[434,4] := 261.9841;
   DATA[434,5] := 8.393553;
   DATA[434,6] := 327.9672;
   DATA[434,7] := 2.439753;
   DATA[434,8] := 2.0;
   DATA[434,9] := 2.0;
   DATA[434,10] := 2.0;
   DATA[434,11] := 19.70357;
   DATA[434,12] := 2.213624;
   DATA[434,13] := 976.9531;
   DATA[434,14] := 1.0;
   DATA[434,15] := 2.0;
   DATA[434,16] := 1.0;
   DATA[434,17] := 1.0;
   DATA[434,18] := 1.0;
   DATA[434,19] := 2.0;
   DATA[434,20] := 148.808;
   DATA[434,21] := 155.96;
   DATA[434,22] := 1.717489;
   DATA[434,23] := 977.5186;
   DATA[434,24] := 2.0;
   DATA[434,25] := 2.0;
   DATA[434,26] := 7.878621;
   DATA[434,27] := 145.1679;
   DATA[434,28] := 263.5863;
   DATA[434,29] := 12.15073;
   DATA[434,30] := 1.728916;
   DATA[434,31] := 1.290765;
   DATA[434,32] := 0.7353967;
   DATA[434,33] := 0.3083624;
   DATA[434,34] := 2.0;
   DATA[434,35] := 250.8652;
   DATA[434,36] := 1.617916;
   DATA[434,37] := 189.727;
   DATA[434,38] := 0.000128152;
   DATA[434,39] := 1.0;
   DATA[435,0] := 2.535631;
   DATA[435,1] := 529.2057;
   DATA[435,2] := 2.0;
   DATA[435,3] := 2.0;
   DATA[435,4] := 261.9841;
   DATA[435,5] := 8.393553;
   DATA[435,6] := 327.9672;
   DATA[435,7] := 2.439753;
   DATA[435,8] := 2.0;
   DATA[435,9] := 2.0;
   DATA[435,10] := 2.0;
   DATA[435,11] := 19.70357;
   DATA[435,12] := 2.213624;
   DATA[435,13] := 976.9931;
   DATA[435,14] := 1.0;
   DATA[435,15] := 2.0;
   DATA[435,16] := 1.0;
   DATA[435,17] := 1.0;
   DATA[435,18] := 1.0;
   DATA[435,19] := 2.0;
   DATA[435,20] := 148.808;
   DATA[435,21] := 155.96;
   DATA[435,22] := 1.717489;
   DATA[435,23] := 977.4802;
   DATA[435,24] := 2.0;
   DATA[435,25] := 2.0;
   DATA[435,26] := 7.878621;
   DATA[435,27] := 145.1679;
   DATA[435,28] := 263.5863;
   DATA[435,29] := 12.15073;
   DATA[435,30] := 1.728916;
   DATA[435,31] := 1.292558;
   DATA[435,32] := 0.7353967;
   DATA[435,33] := 0.3083624;
   DATA[435,34] := 2.0;
   DATA[435,35] := 251.0254;
   DATA[435,36] := 1.617916;
   DATA[435,37] := 189.727;
   DATA[435,38] := 0.000128152;
   DATA[435,39] := 1.0;
   DATA[436,0] := 2.521538;
   DATA[436,1] := 528.3813;
   DATA[436,2] := 2.0;
   DATA[436,3] := 2.0;
   DATA[436,4] := 261.9841;
   DATA[436,5] := 8.393553;
   DATA[436,6] := 328.0954;
   DATA[436,7] := 2.439753;
   DATA[436,8] := 2.0;
   DATA[436,9] := 2.0;
   DATA[436,10] := 2.0;
   DATA[436,11] := 19.70357;
   DATA[436,12] := 2.212087;
   DATA[436,13] := 977.1934;
   DATA[436,14] := 1.0;
   DATA[436,15] := 2.0;
   DATA[436,16] := 1.0;
   DATA[436,17] := 1.0;
   DATA[436,18] := 1.0;
   DATA[436,19] := 2.0;
   DATA[436,20] := 148.808;
   DATA[436,21] := 155.96;
   DATA[436,22] := 1.719284;
   DATA[436,23] := 977.6339;
   DATA[436,24] := 2.0;
   DATA[436,25] := 2.0;
   DATA[436,26] := 7.878621;
   DATA[436,27] := 145.1679;
   DATA[436,28] := 263.5863;
   DATA[436,29] := 12.15073;
   DATA[436,30] := 1.728916;
   DATA[436,31] := 1.302165;
   DATA[436,32] := 0.7353967;
   DATA[436,33] := 0.3083624;
   DATA[436,34] := 2.0;
   DATA[436,35] := 251.0414;
   DATA[436,36] := 1.649953;
   DATA[436,37] := 189.727;
   DATA[436,38] := 0.000128152;
   DATA[436,39] := 1.0;
   DATA[437,0] := 2.503923;
   DATA[437,1] := 528.0281;
   DATA[437,2] := 2.0;
   DATA[437,3] := 2.0;
   DATA[437,4] := 261.9841;
   DATA[437,5] := 8.393553;
   DATA[437,6] := 328.121;
   DATA[437,7] := 2.439753;
   DATA[437,8] := 2.0;
   DATA[437,9] := 2.0;
   DATA[437,10] := 2.0;
   DATA[437,11] := 19.70357;
   DATA[437,12] := 2.212087;
   DATA[437,13] := 977.4738;
   DATA[437,14] := 1.0;
   DATA[437,15] := 2.0;
   DATA[437,16] := 1.0;
   DATA[437,17] := 1.0;
   DATA[437,18] := 1.0;
   DATA[437,19] := 2.0;
   DATA[437,20] := 148.808;
   DATA[437,21] := 155.96;
   DATA[437,22] := 1.719284;
   DATA[437,23] := 977.6339;
   DATA[437,24] := 2.0;
   DATA[437,25] := 2.0;
   DATA[437,26] := 7.878621;
   DATA[437,27] := 145.1166;
   DATA[437,28] := 263.5863;
   DATA[437,29] := 12.15073;
   DATA[437,30] := 1.728916;
   DATA[437,31] := 1.302165;
   DATA[437,32] := 0.7353967;
   DATA[437,33] := 0.3083624;
   DATA[437,34] := 2.0;
   DATA[437,35] := 251.1535;
   DATA[437,36] := 1.69801;
   DATA[437,37] := 189.8071;
   DATA[437,38] := 0.000128152;
   DATA[437,39] := 1.0;
   DATA[438,0] := 2.490472;
   DATA[438,1] := 527.6356;
   DATA[438,2] := 2.0;
   DATA[438,3] := 2.0;
   DATA[438,4] := 262.1764;
   DATA[438,5] := 8.393553;
   DATA[438,6] := 328.121;
   DATA[438,7] := 2.439753;
   DATA[438,8] := 2.0;
   DATA[438,9] := 2.0;
   DATA[438,10] := 2.0;
   DATA[438,11] := 19.61393;
   DATA[438,12] := 2.21119;
   DATA[438,13] := 977.1533;
   DATA[438,14] := 1.0;
   DATA[438,15] := 2.0;
   DATA[438,16] := 1.0;
   DATA[438,17] := 1.0;
   DATA[438,18] := 1.0;
   DATA[438,19] := 2.0;
   DATA[438,20] := 148.808;
   DATA[438,21] := 155.96;
   DATA[438,22] := 1.719284;
   DATA[438,23] := 977.4802;
   DATA[438,24] := 2.0;
   DATA[438,25] := 2.0;
   DATA[438,26] := 7.878621;
   DATA[438,27] := 145.1166;
   DATA[438,28] := 263.362;
   DATA[438,29] := 12.15073;
   DATA[438,30] := 1.731351;
   DATA[438,31] := 1.302165;
   DATA[438,32] := 0.7353967;
   DATA[438,33] := 0.3083624;
   DATA[438,34] := 2.0;
   DATA[438,35] := 251.2817;
   DATA[438,36] := 1.69801;
   DATA[438,37] := 189.9673;
   DATA[438,38] := 0.000128152;
   DATA[438,39] := 1.0;
   DATA[439,0] := 2.473817;
   DATA[439,1] := 527.0861;
   DATA[439,2] := 2.0;
   DATA[439,3] := 2.0;
   DATA[439,4] := 262.1764;
   DATA[439,5] := 8.393553;
   DATA[439,6] := 328.121;
   DATA[439,7] := 2.439753;
   DATA[439,8] := 2.0;
   DATA[439,9] := 2.0;
   DATA[439,10] := 2.0;
   DATA[439,11] := 19.61393;
   DATA[439,12] := 2.210934;
   DATA[439,13] := 976.8729;
   DATA[439,14] := 1.0;
   DATA[439,15] := 2.0;
   DATA[439,16] := 1.0;
   DATA[439,17] := 1.0;
   DATA[439,18] := 1.0;
   DATA[439,19] := 2.0;
   DATA[439,20] := 148.808;
   DATA[439,21] := 155.96;
   DATA[439,22] := 1.719284;
   DATA[439,23] := 977.4802;
   DATA[439,24] := 2.0;
   DATA[439,25] := 2.0;
   DATA[439,26] := 7.878621;
   DATA[439,27] := 145.1166;
   DATA[439,28] := 263.362;
   DATA[439,29] := 12.15073;
   DATA[439,30] := 1.731351;
   DATA[439,31] := 1.302165;
   DATA[439,32] := 0.7353967;
   DATA[439,33] := 0.3083624;
   DATA[439,34] := 2.0;
   DATA[439,35] := 251.2817;
   DATA[439,36] := 1.69801;
   DATA[439,37] := 189.9673;
   DATA[439,38] := 0.000128152;
   DATA[439,39] := 1.0;
   DATA[440,0] := 2.461967;
   DATA[440,1] := 526.4188;
   DATA[440,2] := 2.0;
   DATA[440,3] := 2.0;
   DATA[440,4] := 262.1764;
   DATA[440,5] := 8.393553;
   DATA[440,6] := 328.121;
   DATA[440,7] := 2.439753;
   DATA[440,8] := 2.0;
   DATA[440,9] := 2.0;
   DATA[440,10] := 2.0;
   DATA[440,11] := 19.5435;
   DATA[440,12] := 2.210934;
   DATA[440,13] := 976.8329;
   DATA[440,14] := 1.0;
   DATA[440,15] := 2.0;
   DATA[440,16] := 1.0;
   DATA[440,17] := 1.0;
   DATA[440,18] := 1.0;
   DATA[440,19] := 2.0;
   DATA[440,20] := 148.808;
   DATA[440,21] := 155.96;
   DATA[440,22] := 1.720053;
   DATA[440,23] := 977.4417;
   DATA[440,24] := 2.0;
   DATA[440,25] := 2.0;
   DATA[440,26] := 7.878621;
   DATA[440,27] := 145.1166;
   DATA[440,28] := 263.362;
   DATA[440,29] := 12.15073;
   DATA[440,30] := 1.731351;
   DATA[440,31] := 1.293326;
   DATA[440,32] := 0.7353967;
   DATA[440,33] := 0.3070813;
   DATA[440,34] := 2.0;
   DATA[440,35] := 251.2817;
   DATA[440,36] := 1.69801;
   DATA[440,37] := 189.9673;
   DATA[440,38] := 0.000128152;
   DATA[440,39] := 1.0;
   DATA[441,0] := 2.446594;
   DATA[441,1] := 526.1047;
   DATA[441,2] := 2.0;
   DATA[441,3] := 2.0;
   DATA[441,4] := 262.1764;
   DATA[441,5] := 8.393553;
   DATA[441,6] := 328.121;
   DATA[441,7] := 2.439753;
   DATA[441,8] := 2.0;
   DATA[441,9] := 2.0;
   DATA[441,10] := 2.0;
   DATA[441,11] := 19.5435;
   DATA[441,12] := 2.210934;
   DATA[441,13] := 976.6727;
   DATA[441,14] := 1.0;
   DATA[441,15] := 2.0;
   DATA[441,16] := 1.0;
   DATA[441,17] := 1.0;
   DATA[441,18] := 1.0;
   DATA[441,19] := 2.0;
   DATA[441,20] := 148.808;
   DATA[441,21] := 155.96;
   DATA[441,22] := 1.720565;
   DATA[441,23] := 977.6724;
   DATA[441,24] := 2.0;
   DATA[441,25] := 2.0;
   DATA[441,26] := 7.878621;
   DATA[441,27] := 145.1166;
   DATA[441,28] := 263.362;
   DATA[441,29] := 11.95847;
   DATA[441,30] := 1.731351;
   DATA[441,31] := 1.308185;
   DATA[441,32] := 0.7353967;
   DATA[441,33] := 0.3068251;
   DATA[441,34] := 2.0;
   DATA[441,35] := 251.2817;
   DATA[441,36] := 1.69801;
   DATA[441,37] := 189.9673;
   DATA[441,38] := 0.000128152;
   DATA[441,39] := 1.0;
   DATA[442,0] := 2.425776;
   DATA[442,1] := 526.458;
   DATA[442,2] := 2.0;
   DATA[442,3] := 2.0;
   DATA[442,4] := 262.1764;
   DATA[442,5] := 8.393553;
   DATA[442,6] := 328.121;
   DATA[442,7] := 2.439753;
   DATA[442,8] := 2.0;
   DATA[442,9] := 2.0;
   DATA[442,10] := 2.0;
   DATA[442,11] := 19.5435;
   DATA[442,12] := 2.210934;
   DATA[442,13] := 977.2334;
   DATA[442,14] := 1.0;
   DATA[442,15] := 2.0;
   DATA[442,16] := 1.0;
   DATA[442,17] := 1.0;
   DATA[442,18] := 1.0;
   DATA[442,19] := 2.0;
   DATA[442,20] := 148.808;
   DATA[442,21] := 155.96;
   DATA[442,22] := 1.720565;
   DATA[442,23] := 977.4802;
   DATA[442,24] := 2.0;
   DATA[442,25] := 2.0;
   DATA[442,26] := 7.878621;
   DATA[442,27] := 145.1166;
   DATA[442,28] := 263.362;
   DATA[442,29] := 11.95847;
   DATA[442,30] := 1.731351;
   DATA[442,31] := 1.310747;
   DATA[442,32] := 0.7353967;
   DATA[442,33] := 0.3068251;
   DATA[442,34] := 2.0;
   DATA[442,35] := 251.2817;
   DATA[442,36] := 1.69801;
   DATA[442,37] := 189.9673;
   DATA[442,38] := 0.000128152;
   DATA[442,39] := 1.0;
   DATA[443,0] := 2.420011;
   DATA[443,1] := 527.2038;
   DATA[443,2] := 2.0;
   DATA[443,3] := 2.0;
   DATA[443,4] := 262.1764;
   DATA[443,5] := 8.393553;
   DATA[443,6] := 327.9928;
   DATA[443,7] := 2.439753;
   DATA[443,8] := 2.0;
   DATA[443,9] := 2.0;
   DATA[443,10] := 2.0;
   DATA[443,11] := 19.57232;
   DATA[443,12] := 2.208244;
   DATA[443,13] := 977.0732;
   DATA[443,14] := 1.0;
   DATA[443,15] := 2.0;
   DATA[443,16] := 1.0;
   DATA[443,17] := 1.0;
   DATA[443,18] := 1.0;
   DATA[443,19] := 2.0;
   DATA[443,20] := 148.808;
   DATA[443,21] := 155.96;
   DATA[443,22] := 1.720565;
   DATA[443,23] := 977.7493;
   DATA[443,24] := 2.0;
   DATA[443,25] := 2.0;
   DATA[443,26] := 7.878621;
   DATA[443,27] := 145.1166;
   DATA[443,28] := 263.362;
   DATA[443,29] := 11.95847;
   DATA[443,30] := 1.731351;
   DATA[443,31] := 1.302165;
   DATA[443,32] := 0.7353967;
   DATA[443,33] := 0.3068251;
   DATA[443,34] := 2.0;
   DATA[443,35] := 251.2817;
   DATA[443,36] := 1.69801;
   DATA[443,37] := 189.9673;
   DATA[443,38] := 0.000128152;
   DATA[443,39] := 1.0;
   DATA[444,0] := 2.417769;
   DATA[444,1] := 527.7926;
   DATA[444,2] := 2.0;
   DATA[444,3] := 2.0;
   DATA[444,4] := 262.1764;
   DATA[444,5] := 8.393553;
   DATA[444,6] := 327.9928;
   DATA[444,7] := 2.439753;
   DATA[444,8] := 2.0;
   DATA[444,9] := 2.0;
   DATA[444,10] := 2.0;
   DATA[444,11] := 19.59472;
   DATA[444,12] := 2.207603;
   DATA[444,13] := 976.9931;
   DATA[444,14] := 1.0;
   DATA[444,15] := 2.0;
   DATA[444,16] := 1.0;
   DATA[444,17] := 1.0;
   DATA[444,18] := 1.0;
   DATA[444,19] := 2.0;
   DATA[444,20] := 148.808;
   DATA[444,21] := 155.8575;
   DATA[444,22] := 1.720565;
   DATA[444,23] := 977.7108;
   DATA[444,24] := 2.0;
   DATA[444,25] := 2.0;
   DATA[444,26] := 7.878621;
   DATA[444,27] := 145.1166;
   DATA[444,28] := 263.362;
   DATA[444,29] := 11.95847;
   DATA[444,30] := 1.731351;
   DATA[444,31] := 1.29512;
   DATA[444,32] := 0.7353967;
   DATA[444,33] := 0.3068251;
   DATA[444,34] := 2.0;
   DATA[444,35] := 251.2817;
   DATA[444,36] := 1.69801;
   DATA[444,37] := 189.9673;
   DATA[444,38] := 0.000128152;
   DATA[444,39] := 1.0;
   DATA[445,0] := 2.417769;
   DATA[445,1] := 527.7926;
   DATA[445,2] := 2.0;
   DATA[445,3] := 2.0;
   DATA[445,4] := 262.1764;
   DATA[445,5] := 8.393553;
   DATA[445,6] := 327.9928;
   DATA[445,7] := 2.439753;
   DATA[445,8] := 2.0;
   DATA[445,9] := 2.0;
   DATA[445,10] := 2.0;
   DATA[445,11] := 19.59472;
   DATA[445,12] := 2.206835;
   DATA[445,13] := 977.4337;
   DATA[445,14] := 1.0;
   DATA[445,15] := 2.0;
   DATA[445,16] := 1.0;
   DATA[445,17] := 1.0;
   DATA[445,18] := 1.0;
   DATA[445,19] := 2.0;
   DATA[445,20] := 148.808;
   DATA[445,21] := 155.8318;
   DATA[445,22] := 1.720565;
   DATA[445,23] := 977.557;
   DATA[445,24] := 2.0;
   DATA[445,25] := 2.0;
   DATA[445,26] := 7.878621;
   DATA[445,27] := 145.1166;
   DATA[445,28] := 263.362;
   DATA[445,29] := 11.95847;
   DATA[445,30] := 1.731351;
   DATA[445,31] := 1.291277;
   DATA[445,32] := 0.7353967;
   DATA[445,33] := 0.3068251;
   DATA[445,34] := 2.0;
   DATA[445,35] := 251.2817;
   DATA[445,36] := 1.69801;
   DATA[445,37] := 189.9673;
   DATA[445,38] := 0.000128152;
   DATA[445,39] := 1.0;
   DATA[446,0] := 2.471575;
   DATA[446,1] := 528.2244;
   DATA[446,2] := 2.0;
   DATA[446,3] := 2.0;
   DATA[446,4] := 262.1764;
   DATA[446,5] := 8.393553;
   DATA[446,6] := 327.9928;
   DATA[446,7] := 2.439753;
   DATA[446,8] := 2.0;
   DATA[446,9] := 2.0;
   DATA[446,10] := 2.0;
   DATA[446,11] := 19.59472;
   DATA[446,12] := 2.206835;
   DATA[446,13] := 977.0732;
   DATA[446,14] := 1.0;
   DATA[446,15] := 2.0;
   DATA[446,16] := 1.0;
   DATA[446,17] := 1.0;
   DATA[446,18] := 1.0;
   DATA[446,19] := 2.0;
   DATA[446,20] := 148.808;
   DATA[446,21] := 155.8318;
   DATA[446,22] := 1.719284;
   DATA[446,23] := 977.2879;
   DATA[446,24] := 2.0;
   DATA[446,25] := 2.0;
   DATA[446,26] := 7.878621;
   DATA[446,27] := 145.1166;
   DATA[446,28] := 263.362;
   DATA[446,29] := 11.95847;
   DATA[446,30] := 1.731351;
   DATA[446,31] := 1.291277;
   DATA[446,32] := 0.7353967;
   DATA[446,33] := 0.3068251;
   DATA[446,34] := 2.0;
   DATA[446,35] := 251.2817;
   DATA[446,36] := 1.69801;
   DATA[446,37] := 189.9673;
   DATA[446,38] := 0.000128152;
   DATA[446,39] := 1.0;
   DATA[447,0] := 2.518336;
   DATA[447,1] := 528.5776;
   DATA[447,2] := 2.0;
   DATA[447,3] := 2.0;
   DATA[447,4] := 262.1764;
   DATA[447,5] := 8.393553;
   DATA[447,6] := 327.9928;
   DATA[447,7] := 2.439753;
   DATA[447,8] := 2.0;
   DATA[447,9] := 2.0;
   DATA[447,10] := 2.0;
   DATA[447,11] := 19.66835;
   DATA[447,12] := 2.206835;
   DATA[447,13] := 977.634;
   DATA[447,14] := 1.0;
   DATA[447,15] := 2.0;
   DATA[447,16] := 1.0;
   DATA[447,17] := 1.0;
   DATA[447,18] := 1.0;
   DATA[447,19] := 2.0;
   DATA[447,20] := 148.808;
   DATA[447,21] := 155.8575;
   DATA[447,22] := 1.718771;
   DATA[447,23] := 977.2879;
   DATA[447,24] := 2.0;
   DATA[447,25] := 2.0;
   DATA[447,26] := 7.878621;
   DATA[447,27] := 145.1166;
   DATA[447,28] := 263.362;
   DATA[447,29] := 11.95847;
   DATA[447,30] := 1.731351;
   DATA[447,31] := 1.302037;
   DATA[447,32] := 0.7353967;
   DATA[447,33] := 0.3068251;
   DATA[447,34] := 2.0;
   DATA[447,35] := 251.2817;
   DATA[447,36] := 1.69801;
   DATA[447,37] := 189.9673;
   DATA[447,38] := 0.000128152;
   DATA[447,39] := 1.0;
   DATA[448,0] := 2.558691;
   DATA[448,1] := 529.2057;
   DATA[448,2] := 2.0;
   DATA[448,3] := 2.0;
   DATA[448,4] := 262.1764;
   DATA[448,5] := 8.394835;
   DATA[448,6] := 327.9928;
   DATA[448,7] := 2.439753;
   DATA[448,8] := 2.0;
   DATA[448,9] := 2.0;
   DATA[448,10] := 2.0;
   DATA[448,11] := 19.66835;
   DATA[448,12] := 2.206835;
   DATA[448,13] := 977.7942;
   DATA[448,14] := 1.0;
   DATA[448,15] := 2.0;
   DATA[448,16] := 1.0;
   DATA[448,17] := 1.0;
   DATA[448,18] := 1.0;
   DATA[448,19] := 2.0;
   DATA[448,20] := 148.808;
   DATA[448,21] := 155.96;
   DATA[448,22] := 1.718515;
   DATA[448,23] := 977.0956;
   DATA[448,24] := 2.0;
   DATA[448,25] := 2.0;
   DATA[448,26] := 7.878621;
   DATA[448,27] := 145.1166;
   DATA[448,28] := 263.362;
   DATA[448,29] := 11.95847;
   DATA[448,30] := 1.731351;
   DATA[448,31] := 1.302165;
   DATA[448,32] := 0.7353967;
   DATA[448,33] := 0.3068251;
   DATA[448,34] := 2.0;
   DATA[448,35] := 251.2817;
   DATA[448,36] := 1.69801;
   DATA[448,37] := 189.9673;
   DATA[448,38] := 0.000128152;
   DATA[448,39] := 1.0;
   DATA[449,0] := 2.591679;
   DATA[449,1] := 529.559;
   DATA[449,2] := 2.0;
   DATA[449,3] := 2.0;
   DATA[449,4] := 262.1764;
   DATA[449,5] := 8.395475;
   DATA[449,6] := 328.0185;
   DATA[449,7] := 2.441803;
   DATA[449,8] := 2.0;
   DATA[449,9] := 2.0;
   DATA[449,10] := 2.0;
   DATA[449,11] := 19.66835;
   DATA[449,12] := 2.207731;
   DATA[449,13] := 977.5939;
   DATA[449,14] := 1.0;
   DATA[449,15] := 2.0;
   DATA[449,16] := 1.0;
   DATA[449,17] := 1.0;
   DATA[449,18] := 1.0;
   DATA[449,19] := 2.0;
   DATA[449,20] := 148.808;
   DATA[449,21] := 155.96;
   DATA[449,22] := 1.71813;
   DATA[449,23] := 977.4802;
   DATA[449,24] := 2.0;
   DATA[449,25] := 2.0;
   DATA[449,26] := 7.878621;
   DATA[449,27] := 145.1166;
   DATA[449,28] := 263.362;
   DATA[449,29] := 11.95847;
   DATA[449,30] := 1.731351;
   DATA[449,31] := 1.293839;
   DATA[449,32] := 0.7353967;
   DATA[449,33] := 0.3068251;
   DATA[449,34] := 2.0;
   DATA[449,35] := 251.1535;
   DATA[449,36] := 1.69801;
   DATA[449,37] := 189.9673;
   DATA[449,38] := 0.000128152;
   DATA[449,39] := 1.0;
   DATA[450,0] := 2.631393;
   DATA[450,1] := 529.8337;
   DATA[450,2] := 2.0;
   DATA[450,3] := 2.0;
   DATA[450,4] := 262.1764;
   DATA[450,5] := 8.395475;
   DATA[450,6] := 328.2235;
   DATA[450,7] := 2.442444;
   DATA[450,8] := 2.0;
   DATA[450,9] := 2.0;
   DATA[450,10] := 2.0;
   DATA[450,11] := 19.63954;
   DATA[450,12] := 2.210037;
   DATA[450,13] := 978.0746;
   DATA[450,14] := 1.0;
   DATA[450,15] := 2.0;
   DATA[450,16] := 1.0;
   DATA[450,17] := 1.0;
   DATA[450,18] := 1.0;
   DATA[450,19] := 2.0;
   DATA[450,20] := 148.808;
   DATA[450,21] := 155.96;
   DATA[450,22] := 1.717489;
   DATA[450,23] := 977.7108;
   DATA[450,24] := 2.0;
   DATA[450,25] := 2.0;
   DATA[450,26] := 7.878621;
   DATA[450,27] := 145.1166;
   DATA[450,28] := 263.362;
   DATA[450,29] := 11.95847;
   DATA[450,30] := 1.731351;
   DATA[450,31] := 1.284488;
   DATA[450,32] := 0.7353967;
   DATA[450,33] := 0.3068251;
   DATA[450,34] := 2.0;
   DATA[450,35] := 250.9132;
   DATA[450,36] := 1.69801;
   DATA[450,37] := 189.6469;
   DATA[450,38] := 0.000128152;
   DATA[450,39] := 1.0;
   DATA[451,0] := 2.656375;
   DATA[451,1] := 530.4225;
   DATA[451,2] := 2.0;
   DATA[451,3] := 2.0;
   DATA[451,4] := 262.1764;
   DATA[451,5] := 8.395475;
   DATA[451,6] := 328.2235;
   DATA[451,7] := 2.442444;
   DATA[451,8] := 2.0;
   DATA[451,9] := 2.0;
   DATA[451,10] := 2.0;
   DATA[451,11] := 19.63954;
   DATA[451,12] := 2.210037;
   DATA[451,13] := 978.0746;
   DATA[451,14] := 1.0;
   DATA[451,15] := 2.0;
   DATA[451,16] := 1.0;
   DATA[451,17] := 1.0;
   DATA[451,18] := 1.0;
   DATA[451,19] := 2.0;
   DATA[451,20] := 148.808;
   DATA[451,21] := 155.96;
   DATA[451,22] := 1.715824;
   DATA[451,23] := 977.8646;
   DATA[451,24] := 2.0;
   DATA[451,25] := 2.0;
   DATA[451,26] := 7.878621;
   DATA[451,27] := 145.1166;
   DATA[451,28] := 263.362;
   DATA[451,29] := 11.95847;
   DATA[451,30] := 1.730454;
   DATA[451,31] := 1.274625;
   DATA[451,32] := 0.7353967;
   DATA[451,33] := 0.3080421;
   DATA[451,34] := 2.0;
   DATA[451,35] := 250.9132;
   DATA[451,36] := 1.69801;
   DATA[451,37] := 189.6469;
   DATA[451,38] := 0.000128152;
   DATA[451,39] := 1.0;
   DATA[452,0] := 2.663741;
   DATA[452,1] := 531.3253;
   DATA[452,2] := 2.0;
   DATA[452,3] := 2.0;
   DATA[452,4] := 262.1764;
   DATA[452,5] := 8.395475;
   DATA[452,6] := 328.2235;
   DATA[452,7] := 2.4427;
   DATA[452,8] := 2.0;
   DATA[452,9] := 2.0;
   DATA[452,10] := 2.0;
   DATA[452,11] := 19.64594;
   DATA[452,12] := 2.210037;
   DATA[452,13] := 978.2347;
   DATA[452,14] := 1.0;
   DATA[452,15] := 2.0;
   DATA[452,16] := 1.0;
   DATA[452,17] := 1.0;
   DATA[452,18] := 1.0;
   DATA[452,19] := 2.0;
   DATA[452,20] := 148.808;
   DATA[452,21] := 155.96;
   DATA[452,22] := 1.715824;
   DATA[452,23] := 978.0953;
   DATA[452,24] := 2.0;
   DATA[452,25] := 2.0;
   DATA[452,26] := 7.878621;
   DATA[452,27] := 145.1166;
   DATA[452,28] := 263.362;
   DATA[452,29] := 12.07383;
   DATA[452,30] := 1.728019;
   DATA[452,31] := 1.271935;
   DATA[452,32] := 0.7353967;
   DATA[452,33] := 0.3082983;
   DATA[452,34] := 2.0;
   DATA[452,35] := 250.9132;
   DATA[452,36] := 1.69801;
   DATA[452,37] := 189.4867;
   DATA[452,38] := 0.000128152;
   DATA[452,39] := 1.0;
   DATA[453,0] := 2.657336;
   DATA[453,1] := 531.9926;
   DATA[453,2] := 2.0;
   DATA[453,3] := 2.0;
   DATA[453,4] := 262.1764;
   DATA[453,5] := 8.392271;
   DATA[453,6] := 327.9159;
   DATA[453,7] := 2.4427;
   DATA[453,8] := 2.0;
   DATA[453,9] := 2.0;
   DATA[453,10] := 2.0;
   DATA[453,11] := 19.67155;
   DATA[453,12] := 2.211831;
   DATA[453,13] := 978.3549;
   DATA[453,14] := 1.0;
   DATA[453,15] := 2.0;
   DATA[453,16] := 1.0;
   DATA[453,17] := 1.0;
   DATA[453,18] := 1.0;
   DATA[453,19] := 2.0;
   DATA[453,20] := 148.808;
   DATA[453,21] := 155.96;
   DATA[453,22] := 1.715183;
   DATA[453,23] := 978.0569;
   DATA[453,24] := 2.0;
   DATA[453,25] := 2.0;
   DATA[453,26] := 7.878621;
   DATA[453,27] := 145.1166;
   DATA[453,28] := 263.362;
   DATA[453,29] := 12.11228;
   DATA[453,30] := 1.72725;
   DATA[453,31] := 1.271935;
   DATA[453,32] := 0.7353967;
   DATA[453,33] := 0.3066329;
   DATA[453,34] := 2.0;
   DATA[453,35] := 250.785;
   DATA[453,36] := 1.69801;
   DATA[453,37] := 189.3585;
   DATA[453,38] := 0.000128152;
   DATA[453,39] := 1.0;
   DATA[454,0] := 2.633956;
   DATA[454,1] := 532.6992;
   DATA[454,2] := 2.0;
   DATA[454,3] := 2.0;
   DATA[454,4] := 262.1764;
   DATA[454,5] := 8.392271;
   DATA[454,6] := 327.9159;
   DATA[454,7] := 2.444366;
   DATA[454,8] := 2.0;
   DATA[454,9] := 2.0;
   DATA[454,10] := 2.0;
   DATA[454,11] := 19.67155;
   DATA[454,12] := 2.211831;
   DATA[454,13] := 978.1547;
   DATA[454,14] := 1.0;
   DATA[454,15] := 2.0;
   DATA[454,16] := 1.0;
   DATA[454,17] := 1.0;
   DATA[454,18] := 1.0;
   DATA[454,19] := 2.0;
   DATA[454,20] := 148.808;
   DATA[454,21] := 155.96;
   DATA[454,22] := 1.715183;
   DATA[454,23] := 978.6337;
   DATA[454,24] := 2.0;
   DATA[454,25] := 2.0;
   DATA[454,26] := 7.878621;
   DATA[454,27] := 145.1166;
   DATA[454,28] := 263.362;
   DATA[454,29] := 12.11228;
   DATA[454,30] := 1.726096;
   DATA[454,31] := 1.27232;
   DATA[454,32] := 0.7353967;
   DATA[454,33] := 0.3065689;
   DATA[454,34] := 2.0;
   DATA[454,35] := 250.785;
   DATA[454,36] := 1.69801;
   DATA[454,37] := 189.3585;
   DATA[454,38] := 0.000128152;
   DATA[454,39] := 1.0;
   DATA[455,0] := 2.624027;
   DATA[455,1] := 533.131;
   DATA[455,2] := 2.0;
   DATA[455,3] := 2.0;
   DATA[455,4] := 262.1764;
   DATA[455,5] := 8.392271;
   DATA[455,6] := 327.9159;
   DATA[455,7] := 2.444366;
   DATA[455,8] := 2.0;
   DATA[455,9] := 2.0;
   DATA[455,10] := 2.0;
   DATA[455,11] := 19.67155;
   DATA[455,12] := 2.211831;
   DATA[455,13] := 978.0746;
   DATA[455,14] := 1.0;
   DATA[455,15] := 2.0;
   DATA[455,16] := 1.0;
   DATA[455,17] := 1.0;
   DATA[455,18] := 1.0;
   DATA[455,19] := 2.0;
   DATA[455,20] := 148.808;
   DATA[455,21] := 155.96;
   DATA[455,22] := 1.715183;
   DATA[455,23] := 978.5952;
   DATA[455,24] := 2.0;
   DATA[455,25] := 2.0;
   DATA[455,26] := 7.878621;
   DATA[455,27] := 145.091;
   DATA[455,28] := 263.362;
   DATA[455,29] := 12.11228;
   DATA[455,30] := 1.725327;
   DATA[455,31] := 1.290637;
   DATA[455,32] := 0.7353967;
   DATA[455,33] := 0.3065689;
   DATA[455,34] := 2.0;
   DATA[455,35] := 250.737;
   DATA[455,36] := 1.69801;
   DATA[455,37] := 189.3585;
   DATA[455,38] := 0.000128152;
   DATA[455,39] := 1.0;
   DATA[456,0] := 2.624027;
   DATA[456,1] := 533.7197;
   DATA[456,2] := 2.0;
   DATA[456,3] := 2.0;
   DATA[456,4] := 262.1764;
   DATA[456,5] := 8.392271;
   DATA[456,6] := 327.9159;
   DATA[456,7] := 2.441803;
   DATA[456,8] := 2.0;
   DATA[456,9] := 2.0;
   DATA[456,10] := 2.0;
   DATA[456,11] := 19.67155;
   DATA[456,12] := 2.211959;
   DATA[456,13] := 978.4751;
   DATA[456,14] := 1.0;
   DATA[456,15] := 2.0;
   DATA[456,16] := 1.0;
   DATA[456,17] := 1.0;
   DATA[456,18] := 1.0;
   DATA[456,19] := 2.0;
   DATA[456,20] := 148.808;
   DATA[456,21] := 155.96;
   DATA[456,22] := 1.714798;
   DATA[456,23] := 978.9028;
   DATA[456,24] := 2.0;
   DATA[456,25] := 2.0;
   DATA[456,26] := 7.878621;
   DATA[456,27] := 145.091;
   DATA[456,28] := 263.362;
   DATA[456,29] := 12.11228;
   DATA[456,30] := 1.725327;
   DATA[456,31] := 1.300243;
   DATA[456,32] := 0.7353967;
   DATA[456,33] := 0.3065689;
   DATA[456,34] := 2.0;
   DATA[456,35] := 250.6729;
   DATA[456,36] := 1.69801;
   DATA[456,37] := 189.3585;
   DATA[456,38] := 0.000128152;
   DATA[456,39] := 1.0;
   DATA[457,0] := 2.620504;
   DATA[457,1] := 534.073;
   DATA[457,2] := 2.0;
   DATA[457,3] := 2.0;
   DATA[457,4] := 262.1764;
   DATA[457,5] := 8.392271;
   DATA[457,6] := 327.9159;
   DATA[457,7] := 2.440778;
   DATA[457,8] := 2.0;
   DATA[457,9] := 2.0;
   DATA[457,10] := 2.0;
   DATA[457,11] := 19.67155;
   DATA[457,12] := 2.212984;
   DATA[457,13] := 978.5953;
   DATA[457,14] := 1.0;
   DATA[457,15] := 2.0;
   DATA[457,16] := 1.0;
   DATA[457,17] := 1.0;
   DATA[457,18] := 1.0;
   DATA[457,19] := 2.0;
   DATA[457,20] := 148.808;
   DATA[457,21] := 155.96;
   DATA[457,22] := 1.714798;
   DATA[457,23] := 979.0182;
   DATA[457,24] := 2.0;
   DATA[457,25] := 2.0;
   DATA[457,26] := 7.878621;
   DATA[457,27] := 145.091;
   DATA[457,28] := 263.362;
   DATA[457,29] := 12.11228;
   DATA[457,30] := 1.725327;
   DATA[457,31] := 1.302421;
   DATA[457,32] := 0.7353967;
   DATA[457,33] := 0.3079781;
   DATA[457,34] := 2.0;
   DATA[457,35] := 250.6729;
   DATA[457,36] := 1.69801;
   DATA[457,37] := 189.3585;
   DATA[457,38] := 0.000128152;
   DATA[457,39] := 1.0;
   DATA[458,0] := 2.600006;
   DATA[458,1] := 533.9553;
   DATA[458,2] := 2.0;
   DATA[458,3] := 2.0;
   DATA[458,4] := 262.1764;
   DATA[458,5] := 8.392271;
   DATA[458,6] := 327.9159;
   DATA[458,7] := 2.440521;
   DATA[458,8] := 2.0;
   DATA[458,9] := 2.0;
   DATA[458,10] := 2.0;
   DATA[458,11] := 19.67155;
   DATA[458,12] := 2.212984;
   DATA[458,13] := 979.2361;
   DATA[458,14] := 1.0;
   DATA[458,15] := 2.0;
   DATA[458,16] := 1.0;
   DATA[458,17] := 1.0;
   DATA[458,18] := 1.0;
   DATA[458,19] := 2.0;
   DATA[458,20] := 148.808;
   DATA[458,21] := 155.96;
   DATA[458,22] := 1.717233;
   DATA[458,23] := 979.595;
   DATA[458,24] := 2.0;
   DATA[458,25] := 2.0;
   DATA[458,26] := 7.878621;
   DATA[458,27] := 145.091;
   DATA[458,28] := 263.362;
   DATA[458,29] := 12.11228;
   DATA[458,30] := 1.726096;
   DATA[458,31] := 1.299475;
   DATA[458,32] := 0.7353967;
   DATA[458,33] := 0.3083624;
   DATA[458,34] := 2.0;
   DATA[458,35] := 250.6729;
   DATA[458,36] := 1.69801;
   DATA[458,37] := 189.4066;
   DATA[458,38] := 0.000128152;
   DATA[458,39] := 1.0;
   DATA[459,0] := 2.585914;
   DATA[459,1] := 533.5627;
   DATA[459,2] := 2.0;
   DATA[459,3] := 2.0;
   DATA[459,4] := 262.1764;
   DATA[459,5] := 8.392271;
   DATA[459,6] := 328.1723;
   DATA[459,7] := 2.440521;
   DATA[459,8] := 2.0;
   DATA[459,9] := 2.0;
   DATA[459,10] := 2.0;
   DATA[459,11] := 19.67155;
   DATA[459,12] := 2.209653;
   DATA[459,13] := 979.0759;
   DATA[459,14] := 1.0;
   DATA[459,15] := 2.0;
   DATA[459,16] := 1.0;
   DATA[459,17] := 1.0;
   DATA[459,18] := 1.0;
   DATA[459,19] := 2.0;
   DATA[459,20] := 148.808;
   DATA[459,21] := 155.96;
   DATA[459,22] := 1.717233;
   DATA[459,23] := 979.595;
   DATA[459,24] := 2.0;
   DATA[459,25] := 2.0;
   DATA[459,26] := 7.878621;
   DATA[459,27] := 145.091;
   DATA[459,28] := 263.362;
   DATA[459,29] := 12.11228;
   DATA[459,30] := 1.727378;
   DATA[459,31] := 1.283592;
   DATA[459,32] := 0.7353967;
   DATA[459,33] := 0.3083624;
   DATA[459,34] := 2.0;
   DATA[459,35] := 250.6729;
   DATA[459,36] := 1.69801;
   DATA[459,37] := 189.5988;
   DATA[459,38] := 0.000128152;
   DATA[459,39] := 1.0;
   DATA[460,0] := 2.568299;
   DATA[460,1] := 533.445;
   DATA[460,2] := 2.0;
   DATA[460,3] := 2.0;
   DATA[460,4] := 262.1764;
   DATA[460,5] := 8.392271;
   DATA[460,6] := 328.1723;
   DATA[460,7] := 2.440521;
   DATA[460,8] := 2.0;
   DATA[460,9] := 2.0;
   DATA[460,10] := 2.0;
   DATA[460,11] := 19.62994;
   DATA[460,12] := 2.209653;
   DATA[460,13] := 979.0759;
   DATA[460,14] := 1.0;
   DATA[460,15] := 2.0;
   DATA[460,16] := 1.0;
   DATA[460,17] := 1.0;
   DATA[460,18] := 1.0;
   DATA[460,19] := 2.0;
   DATA[460,20] := 148.808;
   DATA[460,21] := 155.96;
   DATA[460,22] := 1.717233;
   DATA[460,23] := 980.0179;
   DATA[460,24] := 2.0;
   DATA[460,25] := 2.0;
   DATA[460,26] := 7.878621;
   DATA[460,27] := 145.091;
   DATA[460,28] := 263.4581;
   DATA[460,29] := 12.11228;
   DATA[460,30] := 1.727506;
   DATA[460,31] := 1.273345;
   DATA[460,32] := 0.7353967;
   DATA[460,33] := 0.3068251;
   DATA[460,34] := 2.0;
   DATA[460,35] := 250.9773;
   DATA[460,36] := 1.69801;
   DATA[460,37] := 189.6148;
   DATA[460,38] := 0.000128152;
   DATA[460,39] := 1.0;
   DATA[461,0] := 2.556129;
   DATA[461,1] := 533.1702;
   DATA[461,2] := 2.0;
   DATA[461,3] := 2.0;
   DATA[461,4] := 262.1764;
   DATA[461,5] := 8.394835;
   DATA[461,6] := 328.1723;
   DATA[461,7] := 2.440521;
   DATA[461,8] := 2.0;
   DATA[461,9] := 2.0;
   DATA[461,10] := 2.0;
   DATA[461,11] := 19.62994;
   DATA[461,12] := 2.209653;
   DATA[461,13] := 979.156;
   DATA[461,14] := 1.0;
   DATA[461,15] := 2.0;
   DATA[461,16] := 1.0;
   DATA[461,17] := 1.0;
   DATA[461,18] := 1.0;
   DATA[461,19] := 2.0;
   DATA[461,20] := 148.808;
   DATA[461,21] := 155.96;
   DATA[461,22] := 1.717233;
   DATA[461,23] := 980.0179;
   DATA[461,24] := 2.0;
   DATA[461,25] := 2.0;
   DATA[461,26] := 7.878621;
   DATA[461,27] := 145.091;
   DATA[461,28] := 263.4581;
   DATA[461,29] := 12.11228;
   DATA[461,30] := 1.728916;
   DATA[461,31] := 1.271423;
   DATA[461,32] := 0.7353967;
   DATA[461,33] := 0.3068251;
   DATA[461,34] := 2.0;
   DATA[461,35] := 250.9773;
   DATA[461,36] := 1.69801;
   DATA[461,37] := 189.6148;
   DATA[461,38] := 0.000128152;
   DATA[461,39] := 1.0;
   DATA[462,0] := 2.538513;
   DATA[462,1] := 532.8954;
   DATA[462,2] := 2.0;
   DATA[462,3] := 2.0;
   DATA[462,4] := 262.1764;
   DATA[462,5] := 8.394835;
   DATA[462,6] := 327.9928;
   DATA[462,7] := 2.440521;
   DATA[462,8] := 2.0;
   DATA[462,9] := 2.0;
   DATA[462,10] := 2.0;
   DATA[462,11] := 19.73558;
   DATA[462,12] := 2.209653;
   DATA[462,13] := 979.3563;
   DATA[462,14] := 1.0;
   DATA[462,15] := 2.0;
   DATA[462,16] := 1.0;
   DATA[462,17] := 1.0;
   DATA[462,18] := 1.0;
   DATA[462,19] := 2.0;
   DATA[462,20] := 148.808;
   DATA[462,21] := 155.96;
   DATA[462,22] := 1.717105;
   DATA[462,23] := 980.4025;
   DATA[462,24] := 2.0;
   DATA[462,25] := 2.0;
   DATA[462,26] := 7.878621;
   DATA[462,27] := 145.091;
   DATA[462,28] := 263.5222;
   DATA[462,29] := 12.11228;
   DATA[462,30] := 1.728916;
   DATA[462,31] := 1.272064;
   DATA[462,32] := 0.7353967;
   DATA[462,33] := 0.3068251;
   DATA[462,34] := 2.0;
   DATA[462,35] := 250.9773;
   DATA[462,36] := 1.69801;
   DATA[462,37] := 189.6789;
   DATA[462,38] := 0.000128152;
   DATA[462,39] := 1.0;
   DATA[463,0] := 2.52314;
   DATA[463,1] := 533.2487;
   DATA[463,2] := 2.0;
   DATA[463,3] := 2.0;
   DATA[463,4] := 262.1764;
   DATA[463,5] := 8.394835;
   DATA[463,6] := 327.8647;
   DATA[463,7] := 2.440521;
   DATA[463,8] := 2.0;
   DATA[463,9] := 2.0;
   DATA[463,10] := 2.0;
   DATA[463,11] := 19.76439;
   DATA[463,12] := 2.209653;
   DATA[463,13] := 979.2361;
   DATA[463,14] := 1.0;
   DATA[463,15] := 2.0;
   DATA[463,16] := 1.0;
   DATA[463,17] := 1.0;
   DATA[463,18] := 1.0;
   DATA[463,19] := 2.0;
   DATA[463,20] := 148.808;
   DATA[463,21] := 155.96;
   DATA[463,22] := 1.717105;
   DATA[463,23] := 980.1718;
   DATA[463,24] := 2.0;
   DATA[463,25] := 2.0;
   DATA[463,26] := 7.878621;
   DATA[463,27] := 145.091;
   DATA[463,28] := 263.5222;
   DATA[463,29] := 12.11228;
   DATA[463,30] := 1.728916;
   DATA[463,31] := 1.289612;
   DATA[463,32] := 0.7353967;
   DATA[463,33] := 0.3065048;
   DATA[463,34] := 2.0;
   DATA[463,35] := 250.9773;
   DATA[463,36] := 1.69801;
   DATA[463,37] := 189.6789;
   DATA[463,38] := 0.000128152;
   DATA[463,39] := 1.0;
   DATA[464,0] := 2.505845;
   DATA[464,1] := 532.7777;
   DATA[464,2] := 2.0;
   DATA[464,3] := 2.0;
   DATA[464,4] := 262.1764;
   DATA[464,5] := 8.394835;
   DATA[464,6] := 327.8647;
   DATA[464,7] := 2.441675;
   DATA[464,8] := 2.0;
   DATA[464,9] := 2.0;
   DATA[464,10] := 2.0;
   DATA[464,11] := 19.77399;
   DATA[464,12] := 2.209653;
   DATA[464,13] := 978.9958;
   DATA[464,14] := 1.0;
   DATA[464,15] := 2.0;
   DATA[464,16] := 1.0;
   DATA[464,17] := 1.0;
   DATA[464,18] := 1.0;
   DATA[464,19] := 2.0;
   DATA[464,20] := 148.808;
   DATA[464,21] := 155.96;
   DATA[464,22] := 1.717105;
   DATA[464,23] := 980.0564;
   DATA[464,24] := 2.0;
   DATA[464,25] := 2.0;
   DATA[464,26] := 7.878621;
   DATA[464,27] := 145.091;
   DATA[464,28] := 263.5222;
   DATA[464,29] := 12.11228;
   DATA[464,30] := 1.728916;
   DATA[464,31] := 1.292046;
   DATA[464,32] := 0.7353967;
   DATA[464,33] := 0.3065048;
   DATA[464,34] := 2.0;
   DATA[464,35] := 250.9773;
   DATA[464,36] := 1.69801;
   DATA[464,37] := 189.6789;
   DATA[464,38] := 0.000128152;
   DATA[464,39] := 1.0;
   DATA[465,0] := 2.489191;
   DATA[465,1] := 532.5029;
   DATA[465,2] := 2.0;
   DATA[465,3] := 2.0;
   DATA[465,4] := 262.1764;
   DATA[465,5] := 8.394835;
   DATA[465,6] := 327.8647;
   DATA[465,7] := 2.443085;
   DATA[465,8] := 2.0;
   DATA[465,9] := 2.0;
   DATA[465,10] := 2.0;
   DATA[465,11] := 19.7804;
   DATA[465,12] := 2.209653;
   DATA[465,13] := 979.3963;
   DATA[465,14] := 1.0;
   DATA[465,15] := 2.0;
   DATA[465,16] := 1.0;
   DATA[465,17] := 1.0;
   DATA[465,18] := 1.0;
   DATA[465,19] := 2.0;
   DATA[465,20] := 148.808;
   DATA[465,21] := 155.96;
   DATA[465,22] := 1.71813;
   DATA[465,23] := 980.0564;
   DATA[465,24] := 2.0;
   DATA[465,25] := 2.0;
   DATA[465,26] := 7.878621;
   DATA[465,27] := 145.091;
   DATA[465,28] := 263.5222;
   DATA[465,29] := 12.11228;
   DATA[465,30] := 1.728916;
   DATA[465,31] := 1.300243;
   DATA[465,32] := 0.7353967;
   DATA[465,33] := 0.3065048;
   DATA[465,34] := 2.0;
   DATA[465,35] := 251.1215;
   DATA[465,36] := 1.69801;
   DATA[465,37] := 189.8071;
   DATA[465,38] := 0.000128152;
   DATA[465,39] := 1.0;
   DATA[466,0] := 2.47702;
   DATA[466,1] := 531.7964;
   DATA[466,2] := 2.0;
   DATA[466,3] := 2.0;
   DATA[466,4] := 262.1764;
   DATA[466,5] := 8.394835;
   DATA[466,6] := 327.8647;
   DATA[466,7] := 2.443085;
   DATA[466,8] := 2.0;
   DATA[466,9] := 2.0;
   DATA[466,10] := 2.0;
   DATA[466,11] := 19.77079;
   DATA[466,12] := 2.209653;
   DATA[466,13] := 979.9971;
   DATA[466,14] := 1.0;
   DATA[466,15] := 2.0;
   DATA[466,16] := 1.0;
   DATA[466,17] := 1.0;
   DATA[466,18] := 1.0;
   DATA[466,19] := 2.0;
   DATA[466,20] := 148.808;
   DATA[466,21] := 155.96;
   DATA[466,22] := 1.718387;
   DATA[466,23] := 980.1718;
   DATA[466,24] := 2.0;
   DATA[466,25] := 2.0;
   DATA[466,26] := 7.878621;
   DATA[466,27] := 145.091;
   DATA[466,28] := 263.5222;
   DATA[466,29] := 12.11228;
   DATA[466,30] := 1.728916;
   DATA[466,31] := 1.299091;
   DATA[466,32] := 0.7353967;
   DATA[466,33] := 0.3065048;
   DATA[466,34] := 2.0;
   DATA[466,35] := 251.2817;
   DATA[466,36] := 1.69801;
   DATA[466,37] := 190.0154;
   DATA[466,38] := 0.000128152;
   DATA[466,39] := 1.0;
   DATA[467,0] := 2.460366;
   DATA[467,1] := 531.3253;
   DATA[467,2] := 2.0;
   DATA[467,3] := 2.0;
   DATA[467,4] := 262.1764;
   DATA[467,5] := 8.394835;
   DATA[467,6] := 327.8647;
   DATA[467,7] := 2.440521;
   DATA[467,8] := 2.0;
   DATA[467,9] := 2.0;
   DATA[467,10] := 2.0;
   DATA[467,11] := 19.69396;
   DATA[467,12] := 2.213881;
   DATA[467,13] := 980.0372;
   DATA[467,14] := 1.0;
   DATA[467,15] := 2.0;
   DATA[467,16] := 1.0;
   DATA[467,17] := 1.0;
   DATA[467,18] := 1.0;
   DATA[467,19] := 2.0;
   DATA[467,20] := 148.808;
   DATA[467,21] := 155.96;
   DATA[467,22] := 1.720053;
